(* Logix 5000 project; controller reports 1756-L63 rev 20.11; software revision 20.04; part 31 of 52 *)

        [2319].log_data[10].valid := 1, [2319].log_data[11].valid := 1, [2319].log_data[12].valid := 1, [2319].log_data[13].valid := 1, [2319].log_data[14].valid := 1, [2319].log_data[15].valid := 1, [2319].log_data[16].valid := 1, [2319].log_data[17].valid := 1, [2319].log_data[18].valid := 1, [2319].log_data[19].valid := 1, [2319].time.Year := 2023, [2319].time.Month := 1, [2319].time.Day := 17, [2319].time.Hour := 17, [2319].time.Minute := 39, [2319].time.Second := 59, [2320].log_data[0].min := 1.0, [2320].log_data[0].max := 1.0, [2320].log_data[0].total := 300.0, [2320].log_data[0].time := 300.0, [2320].log_data[0].minminute := 40, [2320].log_data[0].maxminute := 40, [2320].log_data[0].valid := 1, [2320].log_data[1].valid := 1, [2320].log_data[2].valid := 1, [2320].log_data[3].valid := 1, [2320].log_data[4].valid := 1, [2320].log_data[5].valid := 1, [2320].log_data[6].valid := 1, [2320].log_data[7].valid := 1, [2320].log_data[8].valid := 1, [2320].log_data[9].valid := 1, [2320].log_data[10].valid := 1, [2320].log_data[11].valid := 1, [2320].log_data[12].valid := 1, [2320].log_data[13].valid := 1, [2320].log_data[14].valid := 1, [2320].log_data[15].valid := 1, [2320].log_data[16].valid := 1, [2320].log_data[17].valid := 1, [2320].log_data[18].valid := 1, [2320].log_data[19].valid := 1, [2320].time.Year := 2023, [2320].time.Month := 1, [2320].time.Day := 17, [2320].time.Hour := 17, [2320].time.Minute := 44, [2320].time.Second := 59, [2321].log_data[0].min := 1.0, [2321].log_data[0].max := 1.0, [2321].log_data[0].total := 300.0, [2321].log_data[0].time := 300.0, [2321].log_data[0].minminute := 45, [2321].log_data[0].maxminute := 45, [2321].log_data[0].valid := 1, [2321].log_data[1].valid := 1, [2321].log_data[2].valid := 1, [2321].log_data[3].valid := 1, [2321].log_data[4].valid := 1, [2321].log_data[5].valid := 1,
        [2321].log_data[6].valid := 1, [2321].log_data[7].valid := 1, [2321].log_data[8].valid := 1, [2321].log_data[9].valid := 1, [2321].log_data[10].valid := 1, [2321].log_data[11].valid := 1, [2321].log_data[12].valid := 1, [2321].log_data[13].valid := 1, [2321].log_data[14].valid := 1, [2321].log_data[15].valid := 1, [2321].log_data[16].valid := 1, [2321].log_data[17].valid := 1, [2321].log_data[18].valid := 1, [2321].log_data[19].valid := 1, [2321].time.Year := 2023, [2321].time.Month := 1, [2321].time.Day := 17, [2321].time.Hour := 17, [2321].time.Minute := 49, [2321].time.Second := 59, [2322].log_data[0].min := 1.0, [2322].log_data[0].max := 1.0, [2322].log_data[0].total := 300.0, [2322].log_data[0].time := 300.0, [2322].log_data[0].minminute := 50, [2322].log_data[0].maxminute := 50, [2322].log_data[0].valid := 1, [2322].log_data[1].valid := 1, [2322].log_data[2].valid := 1, [2322].log_data[3].valid := 1, [2322].log_data[4].valid := 1, [2322].log_data[5].valid := 1, [2322].log_data[6].valid := 1, [2322].log_data[7].valid := 1, [2322].log_data[8].valid := 1, [2322].log_data[9].valid := 1, [2322].log_data[10].valid := 1, [2322].log_data[11].valid := 1, [2322].log_data[12].valid := 1, [2322].log_data[13].valid := 1, [2322].log_data[14].valid := 1, [2322].log_data[15].valid := 1, [2322].log_data[16].valid := 1, [2322].log_data[17].valid := 1, [2322].log_data[18].valid := 1, [2322].log_data[19].valid := 1, [2322].time.Year := 2023, [2322].time.Month := 1, [2322].time.Day := 17, [2322].time.Hour := 17, [2322].time.Minute := 54, [2322].time.Second := 59, [2323].log_data[0].min := 1.0, [2323].log_data[0].max := 1.0, [2323].log_data[0].total := 300.0, [2323].log_data[0].time := 300.0, [2323].log_data[0].minminute := 55, [2323].log_data[0].maxminute := 55, [2323].log_data[0].valid := 1, [2323].log_data[1].valid := 1,
        [2323].log_data[2].valid := 1, [2323].log_data[3].valid := 1, [2323].log_data[4].valid := 1, [2323].log_data[5].valid := 1, [2323].log_data[6].valid := 1, [2323].log_data[7].valid := 1, [2323].log_data[8].valid := 1, [2323].log_data[9].valid := 1, [2323].log_data[10].valid := 1, [2323].log_data[11].valid := 1, [2323].log_data[12].valid := 1, [2323].log_data[13].valid := 1, [2323].log_data[14].valid := 1, [2323].log_data[15].valid := 1, [2323].log_data[16].valid := 1, [2323].log_data[17].valid := 1, [2323].log_data[18].valid := 1, [2323].log_data[19].valid := 1, [2323].time.Year := 2023, [2323].time.Month := 1, [2323].time.Day := 17, [2323].time.Hour := 17, [2323].time.Minute := 59, [2323].time.Second := 59, [2324].log_data[0].min := 1.0, [2324].log_data[0].max := 1.0, [2324].log_data[0].total := 300.0, [2324].log_data[0].time := 300.0, [2324].log_data[0].valid := 1, [2324].log_data[1].valid := 1, [2324].log_data[2].valid := 1, [2324].log_data[3].valid := 1, [2324].log_data[4].valid := 1, [2324].log_data[5].valid := 1, [2324].log_data[6].valid := 1, [2324].log_data[7].valid := 1, [2324].log_data[8].valid := 1, [2324].log_data[9].valid := 1, [2324].log_data[10].valid := 1, [2324].log_data[11].valid := 1, [2324].log_data[12].valid := 1, [2324].log_data[13].valid := 1, [2324].log_data[14].valid := 1, [2324].log_data[15].valid := 1, [2324].log_data[16].valid := 1, [2324].log_data[17].valid := 1, [2324].log_data[18].valid := 1, [2324].log_data[19].valid := 1, [2324].time.Year := 2023, [2324].time.Month := 1, [2324].time.Day := 17, [2324].time.Hour := 18, [2324].time.Minute := 4, [2324].time.Second := 59, [2325].log_data[0].min := 1.0, [2325].log_data[0].max := 1.0, [2325].log_data[0].total := 300.0, [2325].log_data[0].time := 300.0, [2325].log_data[0].minminute := 5, [2325].log_data[0].maxminute := 5,
        [2325].log_data[0].valid := 1, [2325].log_data[1].valid := 1, [2325].log_data[2].valid := 1, [2325].log_data[3].valid := 1, [2325].log_data[4].valid := 1, [2325].log_data[5].valid := 1, [2325].log_data[6].valid := 1, [2325].log_data[7].valid := 1, [2325].log_data[8].valid := 1, [2325].log_data[9].valid := 1, [2325].log_data[10].valid := 1, [2325].log_data[11].valid := 1, [2325].log_data[12].valid := 1, [2325].log_data[13].valid := 1, [2325].log_data[14].valid := 1, [2325].log_data[15].valid := 1, [2325].log_data[16].valid := 1, [2325].log_data[17].valid := 1, [2325].log_data[18].valid := 1, [2325].log_data[19].valid := 1, [2325].time.Year := 2023, [2325].time.Month := 1, [2325].time.Day := 17, [2325].time.Hour := 18, [2325].time.Minute := 9, [2325].time.Second := 59, [2326].log_data[0].min := 1.0, [2326].log_data[0].max := 1.0, [2326].log_data[0].total := 300.0, [2326].log_data[0].time := 300.0, [2326].log_data[0].minminute := 10, [2326].log_data[0].maxminute := 10, [2326].log_data[0].valid := 1, [2326].log_data[1].valid := 1, [2326].log_data[2].valid := 1, [2326].log_data[3].valid := 1, [2326].log_data[4].valid := 1, [2326].log_data[5].valid := 1, [2326].log_data[6].valid := 1, [2326].log_data[7].valid := 1, [2326].log_data[8].valid := 1, [2326].log_data[9].valid := 1, [2326].log_data[10].valid := 1, [2326].log_data[11].valid := 1, [2326].log_data[12].valid := 1, [2326].log_data[13].valid := 1, [2326].log_data[14].valid := 1, [2326].log_data[15].valid := 1, [2326].log_data[16].valid := 1, [2326].log_data[17].valid := 1, [2326].log_data[18].valid := 1, [2326].log_data[19].valid := 1, [2326].time.Year := 2023, [2326].time.Month := 1, [2326].time.Day := 17, [2326].time.Hour := 18, [2326].time.Minute := 14, [2326].time.Second := 59, [2327].log_data[0].min := 1.0, [2327].log_data[0].max := 1.0,
        [2327].log_data[0].total := 300.0, [2327].log_data[0].time := 300.0, [2327].log_data[0].minminute := 15, [2327].log_data[0].maxminute := 15, [2327].log_data[0].valid := 1, [2327].log_data[1].valid := 1, [2327].log_data[2].valid := 1, [2327].log_data[3].valid := 1, [2327].log_data[4].valid := 1, [2327].log_data[5].valid := 1, [2327].log_data[6].valid := 1, [2327].log_data[7].valid := 1, [2327].log_data[8].valid := 1, [2327].log_data[9].valid := 1, [2327].log_data[10].valid := 1, [2327].log_data[11].valid := 1, [2327].log_data[12].valid := 1, [2327].log_data[13].valid := 1, [2327].log_data[14].valid := 1, [2327].log_data[15].valid := 1, [2327].log_data[16].valid := 1, [2327].log_data[17].valid := 1, [2327].log_data[18].valid := 1, [2327].log_data[19].valid := 1, [2327].time.Year := 2023, [2327].time.Month := 1, [2327].time.Day := 17, [2327].time.Hour := 18, [2327].time.Minute := 19, [2327].time.Second := 59, [2328].log_data[0].min := 1.0, [2328].log_data[0].max := 1.0, [2328].log_data[0].total := 300.0, [2328].log_data[0].time := 300.0, [2328].log_data[0].minminute := 20, [2328].log_data[0].maxminute := 20, [2328].log_data[0].valid := 1, [2328].log_data[1].valid := 1, [2328].log_data[2].valid := 1, [2328].log_data[3].valid := 1, [2328].log_data[4].valid := 1, [2328].log_data[5].valid := 1, [2328].log_data[6].valid := 1, [2328].log_data[7].valid := 1, [2328].log_data[8].valid := 1, [2328].log_data[9].valid := 1, [2328].log_data[10].valid := 1, [2328].log_data[11].valid := 1, [2328].log_data[12].valid := 1, [2328].log_data[13].valid := 1, [2328].log_data[14].valid := 1, [2328].log_data[15].valid := 1, [2328].log_data[16].valid := 1, [2328].log_data[17].valid := 1, [2328].log_data[18].valid := 1, [2328].log_data[19].valid := 1, [2328].time.Year := 2023, [2328].time.Month := 1, [2328].time.Day := 17, [2328].time.Hour := 18,
        [2328].time.Minute := 24, [2328].time.Second := 59, [2329].log_data[0].min := 1.0, [2329].log_data[0].max := 1.0, [2329].log_data[0].total := 300.0, [2329].log_data[0].time := 300.0, [2329].log_data[0].minminute := 25, [2329].log_data[0].maxminute := 25, [2329].log_data[0].valid := 1, [2329].log_data[1].valid := 1, [2329].log_data[2].valid := 1, [2329].log_data[3].valid := 1, [2329].log_data[4].valid := 1, [2329].log_data[5].valid := 1, [2329].log_data[6].valid := 1, [2329].log_data[7].valid := 1, [2329].log_data[8].valid := 1, [2329].log_data[9].valid := 1, [2329].log_data[10].valid := 1, [2329].log_data[11].valid := 1, [2329].log_data[12].valid := 1, [2329].log_data[13].valid := 1, [2329].log_data[14].valid := 1, [2329].log_data[15].valid := 1, [2329].log_data[16].valid := 1, [2329].log_data[17].valid := 1, [2329].log_data[18].valid := 1, [2329].log_data[19].valid := 1, [2329].time.Year := 2023, [2329].time.Month := 1, [2329].time.Day := 17, [2329].time.Hour := 18, [2329].time.Minute := 29, [2329].time.Second := 59, [2330].log_data[0].min := 1.0, [2330].log_data[0].max := 1.0, [2330].log_data[0].total := 300.0, [2330].log_data[0].time := 300.0, [2330].log_data[0].minminute := 30, [2330].log_data[0].maxminute := 30, [2330].log_data[0].valid := 1, [2330].log_data[1].valid := 1, [2330].log_data[2].valid := 1, [2330].log_data[3].valid := 1, [2330].log_data[4].valid := 1, [2330].log_data[5].valid := 1, [2330].log_data[6].valid := 1, [2330].log_data[7].valid := 1, [2330].log_data[8].valid := 1, [2330].log_data[9].valid := 1, [2330].log_data[10].valid := 1, [2330].log_data[11].valid := 1, [2330].log_data[12].valid := 1, [2330].log_data[13].valid := 1, [2330].log_data[14].valid := 1, [2330].log_data[15].valid := 1, [2330].log_data[16].valid := 1, [2330].log_data[17].valid := 1, [2330].log_data[18].valid := 1, [2330].log_data[19].valid := 1,
        [2330].time.Year := 2023, [2330].time.Month := 1, [2330].time.Day := 17, [2330].time.Hour := 18, [2330].time.Minute := 34, [2330].time.Second := 59, [2331].log_data[0].min := 1.0, [2331].log_data[0].max := 1.0, [2331].log_data[0].total := 300.0, [2331].log_data[0].time := 300.0, [2331].log_data[0].minminute := 35, [2331].log_data[0].maxminute := 35, [2331].log_data[0].valid := 1, [2331].log_data[1].valid := 1, [2331].log_data[2].valid := 1, [2331].log_data[3].valid := 1, [2331].log_data[4].valid := 1, [2331].log_data[5].valid := 1, [2331].log_data[6].valid := 1, [2331].log_data[7].valid := 1, [2331].log_data[8].valid := 1, [2331].log_data[9].valid := 1, [2331].log_data[10].valid := 1, [2331].log_data[11].valid := 1, [2331].log_data[12].valid := 1, [2331].log_data[13].valid := 1, [2331].log_data[14].valid := 1, [2331].log_data[15].valid := 1, [2331].log_data[16].valid := 1, [2331].log_data[17].valid := 1, [2331].log_data[18].valid := 1, [2331].log_data[19].valid := 1, [2331].time.Year := 2023, [2331].time.Month := 1, [2331].time.Day := 17, [2331].time.Hour := 18, [2331].time.Minute := 39, [2331].time.Second := 59, [2332].log_data[0].min := 1.0, [2332].log_data[0].max := 1.0, [2332].log_data[0].total := 300.0, [2332].log_data[0].time := 300.0, [2332].log_data[0].minminute := 40, [2332].log_data[0].maxminute := 40, [2332].log_data[0].valid := 1, [2332].log_data[1].valid := 1, [2332].log_data[2].valid := 1, [2332].log_data[3].valid := 1, [2332].log_data[4].valid := 1, [2332].log_data[5].valid := 1, [2332].log_data[6].valid := 1, [2332].log_data[7].valid := 1, [2332].log_data[8].valid := 1, [2332].log_data[9].valid := 1, [2332].log_data[10].valid := 1, [2332].log_data[11].valid := 1, [2332].log_data[12].valid := 1, [2332].log_data[13].valid := 1, [2332].log_data[14].valid := 1, [2332].log_data[15].valid := 1,
        [2332].log_data[16].valid := 1, [2332].log_data[17].valid := 1, [2332].log_data[18].valid := 1, [2332].log_data[19].valid := 1, [2332].time.Year := 2023, [2332].time.Month := 1, [2332].time.Day := 17, [2332].time.Hour := 18, [2332].time.Minute := 44, [2332].time.Second := 59, [2333].log_data[0].min := 1.0, [2333].log_data[0].max := 1.0, [2333].log_data[0].total := 300.0, [2333].log_data[0].time := 300.0, [2333].log_data[0].minminute := 45, [2333].log_data[0].maxminute := 45, [2333].log_data[0].valid := 1, [2333].log_data[1].valid := 1, [2333].log_data[2].valid := 1, [2333].log_data[3].valid := 1, [2333].log_data[4].valid := 1, [2333].log_data[5].valid := 1, [2333].log_data[6].valid := 1, [2333].log_data[7].valid := 1, [2333].log_data[8].valid := 1, [2333].log_data[9].valid := 1, [2333].log_data[10].valid := 1, [2333].log_data[11].valid := 1, [2333].log_data[12].valid := 1, [2333].log_data[13].valid := 1, [2333].log_data[14].valid := 1, [2333].log_data[15].valid := 1, [2333].log_data[16].valid := 1, [2333].log_data[17].valid := 1, [2333].log_data[18].valid := 1, [2333].log_data[19].valid := 1, [2333].time.Year := 2023, [2333].time.Month := 1, [2333].time.Day := 17, [2333].time.Hour := 18, [2333].time.Minute := 49, [2333].time.Second := 59, [2334].log_data[0].min := 1.0, [2334].log_data[0].max := 1.0, [2334].log_data[0].total := 300.0, [2334].log_data[0].time := 300.0, [2334].log_data[0].minminute := 50, [2334].log_data[0].maxminute := 50, [2334].log_data[0].valid := 1, [2334].log_data[1].valid := 1, [2334].log_data[2].valid := 1, [2334].log_data[3].valid := 1, [2334].log_data[4].valid := 1, [2334].log_data[5].valid := 1, [2334].log_data[6].valid := 1, [2334].log_data[7].valid := 1, [2334].log_data[8].valid := 1, [2334].log_data[9].valid := 1, [2334].log_data[10].valid := 1, [2334].log_data[11].valid := 1,
        [2334].log_data[12].valid := 1, [2334].log_data[13].valid := 1, [2334].log_data[14].valid := 1, [2334].log_data[15].valid := 1, [2334].log_data[16].valid := 1, [2334].log_data[17].valid := 1, [2334].log_data[18].valid := 1, [2334].log_data[19].valid := 1, [2334].time.Year := 2023, [2334].time.Month := 1, [2334].time.Day := 17, [2334].time.Hour := 18, [2334].time.Minute := 54, [2334].time.Second := 59, [2335].log_data[0].min := 1.0, [2335].log_data[0].max := 1.0, [2335].log_data[0].total := 300.0, [2335].log_data[0].time := 300.0, [2335].log_data[0].minminute := 55, [2335].log_data[0].maxminute := 55, [2335].log_data[0].valid := 1, [2335].log_data[1].valid := 1, [2335].log_data[2].valid := 1, [2335].log_data[3].valid := 1, [2335].log_data[4].valid := 1, [2335].log_data[5].valid := 1, [2335].log_data[6].valid := 1, [2335].log_data[7].valid := 1, [2335].log_data[8].valid := 1, [2335].log_data[9].valid := 1, [2335].log_data[10].valid := 1, [2335].log_data[11].valid := 1, [2335].log_data[12].valid := 1, [2335].log_data[13].valid := 1, [2335].log_data[14].valid := 1, [2335].log_data[15].valid := 1, [2335].log_data[16].valid := 1, [2335].log_data[17].valid := 1, [2335].log_data[18].valid := 1, [2335].log_data[19].valid := 1, [2335].time.Year := 2023, [2335].time.Month := 1, [2335].time.Day := 17, [2335].time.Hour := 18, [2335].time.Minute := 59, [2335].time.Second := 59, [2336].log_data[0].min := 1.0, [2336].log_data[0].max := 1.0, [2336].log_data[0].total := 300.0, [2336].log_data[0].time := 300.0, [2336].log_data[0].valid := 1, [2336].log_data[1].valid := 1, [2336].log_data[2].valid := 1, [2336].log_data[3].valid := 1, [2336].log_data[4].valid := 1, [2336].log_data[5].valid := 1, [2336].log_data[6].valid := 1, [2336].log_data[7].valid := 1, [2336].log_data[8].valid := 1, [2336].log_data[9].valid := 1,
        [2336].log_data[10].valid := 1, [2336].log_data[11].valid := 1, [2336].log_data[12].valid := 1, [2336].log_data[13].valid := 1, [2336].log_data[14].valid := 1, [2336].log_data[15].valid := 1, [2336].log_data[16].valid := 1, [2336].log_data[17].valid := 1, [2336].log_data[18].valid := 1, [2336].log_data[19].valid := 1, [2336].time.Year := 2023, [2336].time.Month := 1, [2336].time.Day := 17, [2336].time.Hour := 19, [2336].time.Minute := 4, [2336].time.Second := 59, [2337].log_data[0].min := 1.0, [2337].log_data[0].max := 1.0, [2337].log_data[0].total := 300.0, [2337].log_data[0].time := 300.0, [2337].log_data[0].minminute := 5, [2337].log_data[0].maxminute := 5, [2337].log_data[0].valid := 1, [2337].log_data[1].valid := 1, [2337].log_data[2].valid := 1, [2337].log_data[3].valid := 1, [2337].log_data[4].valid := 1, [2337].log_data[5].valid := 1, [2337].log_data[6].valid := 1, [2337].log_data[7].valid := 1, [2337].log_data[8].valid := 1, [2337].log_data[9].valid := 1, [2337].log_data[10].valid := 1, [2337].log_data[11].valid := 1, [2337].log_data[12].valid := 1, [2337].log_data[13].valid := 1, [2337].log_data[14].valid := 1, [2337].log_data[15].valid := 1, [2337].log_data[16].valid := 1, [2337].log_data[17].valid := 1, [2337].log_data[18].valid := 1, [2337].log_data[19].valid := 1, [2337].time.Year := 2023, [2337].time.Month := 1, [2337].time.Day := 17, [2337].time.Hour := 19, [2337].time.Minute := 9, [2337].time.Second := 59, [2338].log_data[0].min := 1.0, [2338].log_data[0].max := 1.0, [2338].log_data[0].total := 300.0, [2338].log_data[0].time := 300.0, [2338].log_data[0].minminute := 10, [2338].log_data[0].maxminute := 10, [2338].log_data[0].valid := 1, [2338].log_data[1].valid := 1, [2338].log_data[2].valid := 1, [2338].log_data[3].valid := 1, [2338].log_data[4].valid := 1, [2338].log_data[5].valid := 1,
        [2338].log_data[6].valid := 1, [2338].log_data[7].valid := 1, [2338].log_data[8].valid := 1, [2338].log_data[9].valid := 1, [2338].log_data[10].valid := 1, [2338].log_data[11].valid := 1, [2338].log_data[12].valid := 1, [2338].log_data[13].valid := 1, [2338].log_data[14].valid := 1, [2338].log_data[15].valid := 1, [2338].log_data[16].valid := 1, [2338].log_data[17].valid := 1, [2338].log_data[18].valid := 1, [2338].log_data[19].valid := 1, [2338].time.Year := 2023, [2338].time.Month := 1, [2338].time.Day := 17, [2338].time.Hour := 19, [2338].time.Minute := 14, [2338].time.Second := 59, [2339].log_data[0].min := 1.0, [2339].log_data[0].max := 1.0, [2339].log_data[0].total := 300.0, [2339].log_data[0].time := 300.0, [2339].log_data[0].minminute := 15, [2339].log_data[0].maxminute := 15, [2339].log_data[0].valid := 1, [2339].log_data[1].valid := 1, [2339].log_data[2].valid := 1, [2339].log_data[3].valid := 1, [2339].log_data[4].valid := 1, [2339].log_data[5].valid := 1, [2339].log_data[6].valid := 1, [2339].log_data[7].valid := 1, [2339].log_data[8].valid := 1, [2339].log_data[9].valid := 1, [2339].log_data[10].valid := 1, [2339].log_data[11].valid := 1, [2339].log_data[12].valid := 1, [2339].log_data[13].valid := 1, [2339].log_data[14].valid := 1, [2339].log_data[15].valid := 1, [2339].log_data[16].valid := 1, [2339].log_data[17].valid := 1, [2339].log_data[18].valid := 1, [2339].log_data[19].valid := 1, [2339].time.Year := 2023, [2339].time.Month := 1, [2339].time.Day := 17, [2339].time.Hour := 19, [2339].time.Minute := 19, [2339].time.Second := 59, [2340].log_data[0].min := 1.0, [2340].log_data[0].max := 1.0, [2340].log_data[0].total := 300.0, [2340].log_data[0].time := 300.0, [2340].log_data[0].minminute := 20, [2340].log_data[0].maxminute := 20, [2340].log_data[0].valid := 1, [2340].log_data[1].valid := 1,
        [2340].log_data[2].valid := 1, [2340].log_data[3].valid := 1, [2340].log_data[4].valid := 1, [2340].log_data[5].valid := 1, [2340].log_data[6].valid := 1, [2340].log_data[7].valid := 1, [2340].log_data[8].valid := 1, [2340].log_data[9].valid := 1, [2340].log_data[10].valid := 1, [2340].log_data[11].valid := 1, [2340].log_data[12].valid := 1, [2340].log_data[13].valid := 1, [2340].log_data[14].valid := 1, [2340].log_data[15].valid := 1, [2340].log_data[16].valid := 1, [2340].log_data[17].valid := 1, [2340].log_data[18].valid := 1, [2340].log_data[19].valid := 1, [2340].time.Year := 2023, [2340].time.Month := 1, [2340].time.Day := 17, [2340].time.Hour := 19, [2340].time.Minute := 24, [2340].time.Second := 59, [2341].log_data[0].min := 1.0, [2341].log_data[0].max := 1.0, [2341].log_data[0].total := 300.0, [2341].log_data[0].time := 300.0, [2341].log_data[0].minminute := 25, [2341].log_data[0].maxminute := 25, [2341].log_data[0].valid := 1, [2341].log_data[1].valid := 1, [2341].log_data[2].valid := 1, [2341].log_data[3].valid := 1, [2341].log_data[4].valid := 1, [2341].log_data[5].valid := 1, [2341].log_data[6].valid := 1, [2341].log_data[7].valid := 1, [2341].log_data[8].valid := 1, [2341].log_data[9].valid := 1, [2341].log_data[10].valid := 1, [2341].log_data[11].valid := 1, [2341].log_data[12].valid := 1, [2341].log_data[13].valid := 1, [2341].log_data[14].valid := 1, [2341].log_data[15].valid := 1, [2341].log_data[16].valid := 1, [2341].log_data[17].valid := 1, [2341].log_data[18].valid := 1, [2341].log_data[19].valid := 1, [2341].time.Year := 2023, [2341].time.Month := 1, [2341].time.Day := 17, [2341].time.Hour := 19, [2341].time.Minute := 29, [2341].time.Second := 59, [2342].log_data[0].min := 1.0, [2342].log_data[0].max := 1.0, [2342].log_data[0].total := 300.0, [2342].log_data[0].time := 300.0,
        [2342].log_data[0].minminute := 30, [2342].log_data[0].maxminute := 30, [2342].log_data[0].valid := 1, [2342].log_data[1].valid := 1, [2342].log_data[2].valid := 1, [2342].log_data[3].valid := 1, [2342].log_data[4].valid := 1, [2342].log_data[5].valid := 1, [2342].log_data[6].valid := 1, [2342].log_data[7].valid := 1, [2342].log_data[8].valid := 1, [2342].log_data[9].valid := 1, [2342].log_data[10].valid := 1, [2342].log_data[11].valid := 1, [2342].log_data[12].valid := 1, [2342].log_data[13].valid := 1, [2342].log_data[14].valid := 1, [2342].log_data[15].valid := 1, [2342].log_data[16].valid := 1, [2342].log_data[17].valid := 1, [2342].log_data[18].valid := 1, [2342].log_data[19].valid := 1, [2342].time.Year := 2023, [2342].time.Month := 1, [2342].time.Day := 17, [2342].time.Hour := 19, [2342].time.Minute := 34, [2342].time.Second := 59, [2343].log_data[0].min := 1.0, [2343].log_data[0].max := 1.0, [2343].log_data[0].total := 300.0, [2343].log_data[0].time := 300.0, [2343].log_data[0].minminute := 35, [2343].log_data[0].maxminute := 35, [2343].log_data[0].valid := 1, [2343].log_data[1].valid := 1, [2343].log_data[2].valid := 1, [2343].log_data[3].valid := 1, [2343].log_data[4].valid := 1, [2343].log_data[5].valid := 1, [2343].log_data[6].valid := 1, [2343].log_data[7].valid := 1, [2343].log_data[8].valid := 1, [2343].log_data[9].valid := 1, [2343].log_data[10].valid := 1, [2343].log_data[11].valid := 1, [2343].log_data[12].valid := 1, [2343].log_data[13].valid := 1, [2343].log_data[14].valid := 1, [2343].log_data[15].valid := 1, [2343].log_data[16].valid := 1, [2343].log_data[17].valid := 1, [2343].log_data[18].valid := 1, [2343].log_data[19].valid := 1, [2343].time.Year := 2023, [2343].time.Month := 1, [2343].time.Day := 17, [2343].time.Hour := 19, [2343].time.Minute := 39, [2343].time.Second := 59,
        [2344].log_data[0].min := 1.0, [2344].log_data[0].max := 1.0, [2344].log_data[0].total := 300.0, [2344].log_data[0].time := 300.0, [2344].log_data[0].minminute := 40, [2344].log_data[0].maxminute := 40, [2344].log_data[0].valid := 1, [2344].log_data[1].valid := 1, [2344].log_data[2].valid := 1, [2344].log_data[3].valid := 1, [2344].log_data[4].valid := 1, [2344].log_data[5].valid := 1, [2344].log_data[6].valid := 1, [2344].log_data[7].valid := 1, [2344].log_data[8].valid := 1, [2344].log_data[9].valid := 1, [2344].log_data[10].valid := 1, [2344].log_data[11].valid := 1, [2344].log_data[12].valid := 1, [2344].log_data[13].valid := 1, [2344].log_data[14].valid := 1, [2344].log_data[15].valid := 1, [2344].log_data[16].valid := 1, [2344].log_data[17].valid := 1, [2344].log_data[18].valid := 1, [2344].log_data[19].valid := 1, [2344].time.Year := 2023, [2344].time.Month := 1, [2344].time.Day := 17, [2344].time.Hour := 19, [2344].time.Minute := 44, [2344].time.Second := 59, [2345].log_data[0].min := 1.0, [2345].log_data[0].max := 1.0, [2345].log_data[0].total := 300.0, [2345].log_data[0].time := 300.0, [2345].log_data[0].minminute := 45, [2345].log_data[0].maxminute := 45, [2345].log_data[0].valid := 1, [2345].log_data[1].valid := 1, [2345].log_data[2].valid := 1, [2345].log_data[3].valid := 1, [2345].log_data[4].valid := 1, [2345].log_data[5].valid := 1, [2345].log_data[6].valid := 1, [2345].log_data[7].valid := 1, [2345].log_data[8].valid := 1, [2345].log_data[9].valid := 1, [2345].log_data[10].valid := 1, [2345].log_data[11].valid := 1, [2345].log_data[12].valid := 1, [2345].log_data[13].valid := 1, [2345].log_data[14].valid := 1, [2345].log_data[15].valid := 1, [2345].log_data[16].valid := 1, [2345].log_data[17].valid := 1, [2345].log_data[18].valid := 1, [2345].log_data[19].valid := 1, [2345].time.Year := 2023, [2345].time.Month := 1,
        [2345].time.Day := 17, [2345].time.Hour := 19, [2345].time.Minute := 49, [2345].time.Second := 59, [2346].log_data[0].min := 1.0, [2346].log_data[0].max := 1.0, [2346].log_data[0].total := 300.0, [2346].log_data[0].time := 300.0, [2346].log_data[0].minminute := 50, [2346].log_data[0].maxminute := 50, [2346].log_data[0].valid := 1, [2346].log_data[1].valid := 1, [2346].log_data[2].valid := 1, [2346].log_data[3].valid := 1, [2346].log_data[4].valid := 1, [2346].log_data[5].valid := 1, [2346].log_data[6].valid := 1, [2346].log_data[7].valid := 1, [2346].log_data[8].valid := 1, [2346].log_data[9].valid := 1, [2346].log_data[10].valid := 1, [2346].log_data[11].valid := 1, [2346].log_data[12].valid := 1, [2346].log_data[13].valid := 1, [2346].log_data[14].valid := 1, [2346].log_data[15].valid := 1, [2346].log_data[16].valid := 1, [2346].log_data[17].valid := 1, [2346].log_data[18].valid := 1, [2346].log_data[19].valid := 1, [2346].time.Year := 2023, [2346].time.Month := 1, [2346].time.Day := 17, [2346].time.Hour := 19, [2346].time.Minute := 54, [2346].time.Second := 59, [2347].log_data[0].min := 1.0, [2347].log_data[0].max := 1.0, [2347].log_data[0].total := 300.0, [2347].log_data[0].time := 300.0, [2347].log_data[0].minminute := 55, [2347].log_data[0].maxminute := 55, [2347].log_data[0].valid := 1, [2347].log_data[1].valid := 1, [2347].log_data[2].valid := 1, [2347].log_data[3].valid := 1, [2347].log_data[4].valid := 1, [2347].log_data[5].valid := 1, [2347].log_data[6].valid := 1, [2347].log_data[7].valid := 1, [2347].log_data[8].valid := 1, [2347].log_data[9].valid := 1, [2347].log_data[10].valid := 1, [2347].log_data[11].valid := 1, [2347].log_data[12].valid := 1, [2347].log_data[13].valid := 1, [2347].log_data[14].valid := 1, [2347].log_data[15].valid := 1, [2347].log_data[16].valid := 1, [2347].log_data[17].valid := 1,
        [2347].log_data[18].valid := 1, [2347].log_data[19].valid := 1, [2347].time.Year := 2023, [2347].time.Month := 1, [2347].time.Day := 17, [2347].time.Hour := 19, [2347].time.Minute := 59, [2347].time.Second := 59, [2348].log_data[0].min := 1.0, [2348].log_data[0].max := 1.0, [2348].log_data[0].total := 299.5, [2348].log_data[0].time := 299.5, [2348].log_data[0].valid := 1, [2348].log_data[1].valid := 1, [2348].log_data[2].valid := 1, [2348].log_data[3].valid := 1, [2348].log_data[4].valid := 1, [2348].log_data[5].valid := 1, [2348].log_data[6].valid := 1, [2348].log_data[7].valid := 1, [2348].log_data[8].valid := 1, [2348].log_data[9].valid := 1, [2348].log_data[10].valid := 1, [2348].log_data[11].valid := 1, [2348].log_data[12].valid := 1, [2348].log_data[13].valid := 1, [2348].log_data[14].valid := 1, [2348].log_data[15].valid := 1, [2348].log_data[16].valid := 1, [2348].log_data[17].valid := 1, [2348].log_data[18].valid := 1, [2348].log_data[19].valid := 1, [2348].time.Year := 2023, [2348].time.Month := 1, [2348].time.Day := 17, [2348].time.Hour := 20, [2348].time.Minute := 4, [2348].time.Second := 59, [2349].log_data[0].min := 1.0, [2349].log_data[0].max := 1.0, [2349].log_data[0].total := 300.0, [2349].log_data[0].time := 300.0, [2349].log_data[0].minminute := 5, [2349].log_data[0].maxminute := 5, [2349].log_data[0].valid := 1, [2349].log_data[1].valid := 1, [2349].log_data[2].valid := 1, [2349].log_data[3].valid := 1, [2349].log_data[4].valid := 1, [2349].log_data[5].valid := 1, [2349].log_data[6].valid := 1, [2349].log_data[7].valid := 1, [2349].log_data[8].valid := 1, [2349].log_data[9].valid := 1, [2349].log_data[10].valid := 1, [2349].log_data[11].valid := 1, [2349].log_data[12].valid := 1, [2349].log_data[13].valid := 1, [2349].log_data[14].valid := 1, [2349].log_data[15].valid := 1,
        [2349].log_data[16].valid := 1, [2349].log_data[17].valid := 1, [2349].log_data[18].valid := 1, [2349].log_data[19].valid := 1, [2349].time.Year := 2023, [2349].time.Month := 1, [2349].time.Day := 17, [2349].time.Hour := 20, [2349].time.Minute := 9, [2349].time.Second := 59, [2350].log_data[0].min := 1.0, [2350].log_data[0].max := 1.0, [2350].log_data[0].total := 300.0, [2350].log_data[0].time := 300.0, [2350].log_data[0].minminute := 10, [2350].log_data[0].maxminute := 10, [2350].log_data[0].valid := 1, [2350].log_data[1].valid := 1, [2350].log_data[2].valid := 1, [2350].log_data[3].valid := 1, [2350].log_data[4].valid := 1, [2350].log_data[5].valid := 1, [2350].log_data[6].valid := 1, [2350].log_data[7].valid := 1, [2350].log_data[8].valid := 1, [2350].log_data[9].valid := 1, [2350].log_data[10].valid := 1, [2350].log_data[11].valid := 1, [2350].log_data[12].valid := 1, [2350].log_data[13].valid := 1, [2350].log_data[14].valid := 1, [2350].log_data[15].valid := 1, [2350].log_data[16].valid := 1, [2350].log_data[17].valid := 1, [2350].log_data[18].valid := 1, [2350].log_data[19].valid := 1, [2350].time.Year := 2023, [2350].time.Month := 1, [2350].time.Day := 17, [2350].time.Hour := 20, [2350].time.Minute := 14, [2350].time.Second := 59, [2351].log_data[0].min := 1.0, [2351].log_data[0].max := 1.0, [2351].log_data[0].total := 300.0, [2351].log_data[0].time := 300.0, [2351].log_data[0].minminute := 15, [2351].log_data[0].maxminute := 15, [2351].log_data[0].valid := 1, [2351].log_data[1].valid := 1, [2351].log_data[2].valid := 1, [2351].log_data[3].valid := 1, [2351].log_data[4].valid := 1, [2351].log_data[5].valid := 1, [2351].log_data[6].valid := 1, [2351].log_data[7].valid := 1, [2351].log_data[8].valid := 1, [2351].log_data[9].valid := 1, [2351].log_data[10].valid := 1, [2351].log_data[11].valid := 1,
        [2351].log_data[12].valid := 1, [2351].log_data[13].valid := 1, [2351].log_data[14].valid := 1, [2351].log_data[15].valid := 1, [2351].log_data[16].valid := 1, [2351].log_data[17].valid := 1, [2351].log_data[18].valid := 1, [2351].log_data[19].valid := 1, [2351].time.Year := 2023, [2351].time.Month := 1, [2351].time.Day := 17, [2351].time.Hour := 20, [2351].time.Minute := 19, [2351].time.Second := 59, [2352].log_data[0].min := 1.0, [2352].log_data[0].max := 1.0, [2352].log_data[0].total := 300.0, [2352].log_data[0].time := 300.0, [2352].log_data[0].minminute := 20, [2352].log_data[0].maxminute := 20, [2352].log_data[0].valid := 1, [2352].log_data[1].valid := 1, [2352].log_data[2].valid := 1, [2352].log_data[3].valid := 1, [2352].log_data[4].valid := 1, [2352].log_data[5].valid := 1, [2352].log_data[6].valid := 1, [2352].log_data[7].valid := 1, [2352].log_data[8].valid := 1, [2352].log_data[9].valid := 1, [2352].log_data[10].valid := 1, [2352].log_data[11].valid := 1, [2352].log_data[12].valid := 1, [2352].log_data[13].valid := 1, [2352].log_data[14].valid := 1, [2352].log_data[15].valid := 1, [2352].log_data[16].valid := 1, [2352].log_data[17].valid := 1, [2352].log_data[18].valid := 1, [2352].log_data[19].valid := 1, [2352].time.Year := 2023, [2352].time.Month := 1, [2352].time.Day := 17, [2352].time.Hour := 20, [2352].time.Minute := 24, [2352].time.Second := 59, [2353].log_data[0].min := 1.0, [2353].log_data[0].max := 1.0, [2353].log_data[0].total := 300.0, [2353].log_data[0].time := 300.0, [2353].log_data[0].minminute := 25, [2353].log_data[0].maxminute := 25, [2353].log_data[0].valid := 1, [2353].log_data[1].valid := 1, [2353].log_data[2].valid := 1, [2353].log_data[3].valid := 1, [2353].log_data[4].valid := 1, [2353].log_data[5].valid := 1, [2353].log_data[6].valid := 1, [2353].log_data[7].valid := 1,
        [2353].log_data[8].valid := 1, [2353].log_data[9].valid := 1, [2353].log_data[10].valid := 1, [2353].log_data[11].valid := 1, [2353].log_data[12].valid := 1, [2353].log_data[13].valid := 1, [2353].log_data[14].valid := 1, [2353].log_data[15].valid := 1, [2353].log_data[16].valid := 1, [2353].log_data[17].valid := 1, [2353].log_data[18].valid := 1, [2353].log_data[19].valid := 1, [2353].time.Year := 2023, [2353].time.Month := 1, [2353].time.Day := 17, [2353].time.Hour := 20, [2353].time.Minute := 29, [2353].time.Second := 59, [2354].log_data[0].min := 1.0, [2354].log_data[0].max := 1.0, [2354].log_data[0].total := 300.0, [2354].log_data[0].time := 300.0, [2354].log_data[0].minminute := 30, [2354].log_data[0].maxminute := 30, [2354].log_data[0].valid := 1, [2354].log_data[1].valid := 1, [2354].log_data[2].valid := 1, [2354].log_data[3].valid := 1, [2354].log_data[4].valid := 1, [2354].log_data[5].valid := 1, [2354].log_data[6].valid := 1, [2354].log_data[7].valid := 1, [2354].log_data[8].valid := 1, [2354].log_data[9].valid := 1, [2354].log_data[10].valid := 1, [2354].log_data[11].valid := 1, [2354].log_data[12].valid := 1, [2354].log_data[13].valid := 1, [2354].log_data[14].valid := 1, [2354].log_data[15].valid := 1, [2354].log_data[16].valid := 1, [2354].log_data[17].valid := 1, [2354].log_data[18].valid := 1, [2354].log_data[19].valid := 1, [2354].time.Year := 2023, [2354].time.Month := 1, [2354].time.Day := 17, [2354].time.Hour := 20, [2354].time.Minute := 34, [2354].time.Second := 59, [2355].log_data[0].min := 1.0, [2355].log_data[0].max := 1.0, [2355].log_data[0].total := 300.0, [2355].log_data[0].time := 300.0, [2355].log_data[0].minminute := 35, [2355].log_data[0].maxminute := 35, [2355].log_data[0].valid := 1, [2355].log_data[1].valid := 1, [2355].log_data[2].valid := 1, [2355].log_data[3].valid := 1,
        [2355].log_data[4].valid := 1, [2355].log_data[5].valid := 1, [2355].log_data[6].valid := 1, [2355].log_data[7].valid := 1, [2355].log_data[8].valid := 1, [2355].log_data[9].valid := 1, [2355].log_data[10].valid := 1, [2355].log_data[11].valid := 1, [2355].log_data[12].valid := 1, [2355].log_data[13].valid := 1, [2355].log_data[14].valid := 1, [2355].log_data[15].valid := 1, [2355].log_data[16].valid := 1, [2355].log_data[17].valid := 1, [2355].log_data[18].valid := 1, [2355].log_data[19].valid := 1, [2355].time.Year := 2023, [2355].time.Month := 1, [2355].time.Day := 17, [2355].time.Hour := 20, [2355].time.Minute := 39, [2355].time.Second := 59, [2356].log_data[0].min := 1.0, [2356].log_data[0].max := 1.0, [2356].log_data[0].total := 300.0, [2356].log_data[0].time := 300.0, [2356].log_data[0].minminute := 40, [2356].log_data[0].maxminute := 40, [2356].log_data[0].valid := 1, [2356].log_data[1].valid := 1, [2356].log_data[2].valid := 1, [2356].log_data[3].valid := 1, [2356].log_data[4].valid := 1, [2356].log_data[5].valid := 1, [2356].log_data[6].valid := 1, [2356].log_data[7].valid := 1, [2356].log_data[8].valid := 1, [2356].log_data[9].valid := 1, [2356].log_data[10].valid := 1, [2356].log_data[11].valid := 1, [2356].log_data[12].valid := 1, [2356].log_data[13].valid := 1, [2356].log_data[14].valid := 1, [2356].log_data[15].valid := 1, [2356].log_data[16].valid := 1, [2356].log_data[17].valid := 1, [2356].log_data[18].valid := 1, [2356].log_data[19].valid := 1, [2356].time.Year := 2023, [2356].time.Month := 1, [2356].time.Day := 17, [2356].time.Hour := 20, [2356].time.Minute := 44, [2356].time.Second := 59, [2357].log_data[0].min := 1.0, [2357].log_data[0].max := 1.0, [2357].log_data[0].total := 300.0, [2357].log_data[0].time := 300.0, [2357].log_data[0].minminute := 45, [2357].log_data[0].maxminute := 45,
        [2357].log_data[0].valid := 1, [2357].log_data[1].valid := 1, [2357].log_data[2].valid := 1, [2357].log_data[3].valid := 1, [2357].log_data[4].valid := 1, [2357].log_data[5].valid := 1, [2357].log_data[6].valid := 1, [2357].log_data[7].valid := 1, [2357].log_data[8].valid := 1, [2357].log_data[9].valid := 1, [2357].log_data[10].valid := 1, [2357].log_data[11].valid := 1, [2357].log_data[12].valid := 1, [2357].log_data[13].valid := 1, [2357].log_data[14].valid := 1, [2357].log_data[15].valid := 1, [2357].log_data[16].valid := 1, [2357].log_data[17].valid := 1, [2357].log_data[18].valid := 1, [2357].log_data[19].valid := 1, [2357].time.Year := 2023, [2357].time.Month := 1, [2357].time.Day := 17, [2357].time.Hour := 20, [2357].time.Minute := 49, [2357].time.Second := 59, [2358].log_data[0].min := 1.0, [2358].log_data[0].max := 1.0, [2358].log_data[0].total := 300.0, [2358].log_data[0].time := 300.0, [2358].log_data[0].minminute := 50, [2358].log_data[0].maxminute := 50, [2358].log_data[0].valid := 1, [2358].log_data[1].valid := 1, [2358].log_data[2].valid := 1, [2358].log_data[3].valid := 1, [2358].log_data[4].valid := 1, [2358].log_data[5].valid := 1, [2358].log_data[6].valid := 1, [2358].log_data[7].valid := 1, [2358].log_data[8].valid := 1, [2358].log_data[9].valid := 1, [2358].log_data[10].valid := 1, [2358].log_data[11].valid := 1, [2358].log_data[12].valid := 1, [2358].log_data[13].valid := 1, [2358].log_data[14].valid := 1, [2358].log_data[15].valid := 1, [2358].log_data[16].valid := 1, [2358].log_data[17].valid := 1, [2358].log_data[18].valid := 1, [2358].log_data[19].valid := 1, [2358].time.Year := 2023, [2358].time.Month := 1, [2358].time.Day := 17, [2358].time.Hour := 20, [2358].time.Minute := 54, [2358].time.Second := 59, [2359].log_data[0].min := 1.0, [2359].log_data[0].max := 1.0,
        [2359].log_data[0].total := 300.0, [2359].log_data[0].time := 300.0, [2359].log_data[0].minminute := 55, [2359].log_data[0].maxminute := 55, [2359].log_data[0].valid := 1, [2359].log_data[1].valid := 1, [2359].log_data[2].valid := 1, [2359].log_data[3].valid := 1, [2359].log_data[4].valid := 1, [2359].log_data[5].valid := 1, [2359].log_data[6].valid := 1, [2359].log_data[7].valid := 1, [2359].log_data[8].valid := 1, [2359].log_data[9].valid := 1, [2359].log_data[10].valid := 1, [2359].log_data[11].valid := 1, [2359].log_data[12].valid := 1, [2359].log_data[13].valid := 1, [2359].log_data[14].valid := 1, [2359].log_data[15].valid := 1, [2359].log_data[16].valid := 1, [2359].log_data[17].valid := 1, [2359].log_data[18].valid := 1, [2359].log_data[19].valid := 1, [2359].time.Year := 2023, [2359].time.Month := 1, [2359].time.Day := 17, [2359].time.Hour := 20, [2359].time.Minute := 59, [2359].time.Second := 59, [2360].log_data[0].min := 1.0, [2360].log_data[0].max := 1.0, [2360].log_data[0].total := 300.0, [2360].log_data[0].time := 300.0, [2360].log_data[0].valid := 1, [2360].log_data[1].valid := 1, [2360].log_data[2].valid := 1, [2360].log_data[3].valid := 1, [2360].log_data[4].valid := 1, [2360].log_data[5].valid := 1, [2360].log_data[6].valid := 1, [2360].log_data[7].valid := 1, [2360].log_data[8].valid := 1, [2360].log_data[9].valid := 1, [2360].log_data[10].valid := 1, [2360].log_data[11].valid := 1, [2360].log_data[12].valid := 1, [2360].log_data[13].valid := 1, [2360].log_data[14].valid := 1, [2360].log_data[15].valid := 1, [2360].log_data[16].valid := 1, [2360].log_data[17].valid := 1, [2360].log_data[18].valid := 1, [2360].log_data[19].valid := 1, [2360].time.Year := 2023, [2360].time.Month := 1, [2360].time.Day := 17, [2360].time.Hour := 21, [2360].time.Minute := 4, [2360].time.Second := 59,
        [2361].log_data[0].min := 1.0, [2361].log_data[0].max := 1.0, [2361].log_data[0].total := 300.0, [2361].log_data[0].time := 300.0, [2361].log_data[0].minminute := 5, [2361].log_data[0].maxminute := 5, [2361].log_data[0].valid := 1, [2361].log_data[1].valid := 1, [2361].log_data[2].valid := 1, [2361].log_data[3].valid := 1, [2361].log_data[4].valid := 1, [2361].log_data[5].valid := 1, [2361].log_data[6].valid := 1, [2361].log_data[7].valid := 1, [2361].log_data[8].valid := 1, [2361].log_data[9].valid := 1, [2361].log_data[10].valid := 1, [2361].log_data[11].valid := 1, [2361].log_data[12].valid := 1, [2361].log_data[13].valid := 1, [2361].log_data[14].valid := 1, [2361].log_data[15].valid := 1, [2361].log_data[16].valid := 1, [2361].log_data[17].valid := 1, [2361].log_data[18].valid := 1, [2361].log_data[19].valid := 1, [2361].time.Year := 2023, [2361].time.Month := 1, [2361].time.Day := 17, [2361].time.Hour := 21, [2361].time.Minute := 9, [2361].time.Second := 59, [2362].log_data[0].min := 1.0, [2362].log_data[0].max := 1.0, [2362].log_data[0].total := 300.0, [2362].log_data[0].time := 300.0, [2362].log_data[0].minminute := 10, [2362].log_data[0].maxminute := 10, [2362].log_data[0].valid := 1, [2362].log_data[1].valid := 1, [2362].log_data[2].valid := 1, [2362].log_data[3].valid := 1, [2362].log_data[4].valid := 1, [2362].log_data[5].valid := 1, [2362].log_data[6].valid := 1, [2362].log_data[7].valid := 1, [2362].log_data[8].valid := 1, [2362].log_data[9].valid := 1, [2362].log_data[10].valid := 1, [2362].log_data[11].valid := 1, [2362].log_data[12].valid := 1, [2362].log_data[13].valid := 1, [2362].log_data[14].valid := 1, [2362].log_data[15].valid := 1, [2362].log_data[16].valid := 1, [2362].log_data[17].valid := 1, [2362].log_data[18].valid := 1, [2362].log_data[19].valid := 1, [2362].time.Year := 2023, [2362].time.Month := 1,
        [2362].time.Day := 17, [2362].time.Hour := 21, [2362].time.Minute := 14, [2362].time.Second := 59, [2363].log_data[0].min := 1.0, [2363].log_data[0].max := 1.0, [2363].log_data[0].total := 300.0, [2363].log_data[0].time := 300.0, [2363].log_data[0].minminute := 15, [2363].log_data[0].maxminute := 15, [2363].log_data[0].valid := 1, [2363].log_data[1].valid := 1, [2363].log_data[2].valid := 1, [2363].log_data[3].valid := 1, [2363].log_data[4].valid := 1, [2363].log_data[5].valid := 1, [2363].log_data[6].valid := 1, [2363].log_data[7].valid := 1, [2363].log_data[8].valid := 1, [2363].log_data[9].valid := 1, [2363].log_data[10].valid := 1, [2363].log_data[11].valid := 1, [2363].log_data[12].valid := 1, [2363].log_data[13].valid := 1, [2363].log_data[14].valid := 1, [2363].log_data[15].valid := 1, [2363].log_data[16].valid := 1, [2363].log_data[17].valid := 1, [2363].log_data[18].valid := 1, [2363].log_data[19].valid := 1, [2363].time.Year := 2023, [2363].time.Month := 1, [2363].time.Day := 17, [2363].time.Hour := 21, [2363].time.Minute := 19, [2363].time.Second := 59, [2364].log_data[0].min := 1.0, [2364].log_data[0].max := 1.0, [2364].log_data[0].total := 300.0, [2364].log_data[0].time := 300.0, [2364].log_data[0].minminute := 20, [2364].log_data[0].maxminute := 20, [2364].log_data[0].valid := 1, [2364].log_data[1].valid := 1, [2364].log_data[2].valid := 1, [2364].log_data[3].valid := 1, [2364].log_data[4].valid := 1, [2364].log_data[5].valid := 1, [2364].log_data[6].valid := 1, [2364].log_data[7].valid := 1, [2364].log_data[8].valid := 1, [2364].log_data[9].valid := 1, [2364].log_data[10].valid := 1, [2364].log_data[11].valid := 1, [2364].log_data[12].valid := 1, [2364].log_data[13].valid := 1, [2364].log_data[14].valid := 1, [2364].log_data[15].valid := 1, [2364].log_data[16].valid := 1, [2364].log_data[17].valid := 1,
        [2364].log_data[18].valid := 1, [2364].log_data[19].valid := 1, [2364].time.Year := 2023, [2364].time.Month := 1, [2364].time.Day := 17, [2364].time.Hour := 21, [2364].time.Minute := 24, [2364].time.Second := 59, [2365].log_data[0].min := 1.0, [2365].log_data[0].max := 1.0, [2365].log_data[0].total := 300.0, [2365].log_data[0].time := 300.0, [2365].log_data[0].minminute := 25, [2365].log_data[0].maxminute := 25, [2365].log_data[0].valid := 1, [2365].log_data[1].valid := 1, [2365].log_data[2].valid := 1, [2365].log_data[3].valid := 1, [2365].log_data[4].valid := 1, [2365].log_data[5].valid := 1, [2365].log_data[6].valid := 1, [2365].log_data[7].valid := 1, [2365].log_data[8].valid := 1, [2365].log_data[9].valid := 1, [2365].log_data[10].valid := 1, [2365].log_data[11].valid := 1, [2365].log_data[12].valid := 1, [2365].log_data[13].valid := 1, [2365].log_data[14].valid := 1, [2365].log_data[15].valid := 1, [2365].log_data[16].valid := 1, [2365].log_data[17].valid := 1, [2365].log_data[18].valid := 1, [2365].log_data[19].valid := 1, [2365].time.Year := 2023, [2365].time.Month := 1, [2365].time.Day := 17, [2365].time.Hour := 21, [2365].time.Minute := 29, [2365].time.Second := 59, [2366].log_data[0].min := 1.0, [2366].log_data[0].max := 1.0, [2366].log_data[0].total := 300.0, [2366].log_data[0].time := 300.0, [2366].log_data[0].minminute := 30, [2366].log_data[0].maxminute := 30, [2366].log_data[0].valid := 1, [2366].log_data[1].valid := 1, [2366].log_data[2].valid := 1, [2366].log_data[3].valid := 1, [2366].log_data[4].valid := 1, [2366].log_data[5].valid := 1, [2366].log_data[6].valid := 1, [2366].log_data[7].valid := 1, [2366].log_data[8].valid := 1, [2366].log_data[9].valid := 1, [2366].log_data[10].valid := 1, [2366].log_data[11].valid := 1, [2366].log_data[12].valid := 1, [2366].log_data[13].valid := 1,
        [2366].log_data[14].valid := 1, [2366].log_data[15].valid := 1, [2366].log_data[16].valid := 1, [2366].log_data[17].valid := 1, [2366].log_data[18].valid := 1, [2366].log_data[19].valid := 1, [2366].time.Year := 2023, [2366].time.Month := 1, [2366].time.Day := 17, [2366].time.Hour := 21, [2366].time.Minute := 34, [2366].time.Second := 59, [2367].log_data[0].min := 1.0, [2367].log_data[0].max := 1.0, [2367].log_data[0].total := 300.0, [2367].log_data[0].time := 300.0, [2367].log_data[0].minminute := 35, [2367].log_data[0].maxminute := 35, [2367].log_data[0].valid := 1, [2367].log_data[1].valid := 1, [2367].log_data[2].valid := 1, [2367].log_data[3].valid := 1, [2367].log_data[4].valid := 1, [2367].log_data[5].valid := 1, [2367].log_data[6].valid := 1, [2367].log_data[7].valid := 1, [2367].log_data[8].valid := 1, [2367].log_data[9].valid := 1, [2367].log_data[10].valid := 1, [2367].log_data[11].valid := 1, [2367].log_data[12].valid := 1, [2367].log_data[13].valid := 1, [2367].log_data[14].valid := 1, [2367].log_data[15].valid := 1, [2367].log_data[16].valid := 1, [2367].log_data[17].valid := 1, [2367].log_data[18].valid := 1, [2367].log_data[19].valid := 1, [2367].time.Year := 2023, [2367].time.Month := 1, [2367].time.Day := 17, [2367].time.Hour := 21, [2367].time.Minute := 39, [2367].time.Second := 59, [2368].log_data[0].min := 1.0, [2368].log_data[0].max := 1.0, [2368].log_data[0].total := 300.0, [2368].log_data[0].time := 300.0, [2368].log_data[0].minminute := 40, [2368].log_data[0].maxminute := 40, [2368].log_data[0].valid := 1, [2368].log_data[1].valid := 1, [2368].log_data[2].valid := 1, [2368].log_data[3].valid := 1, [2368].log_data[4].valid := 1, [2368].log_data[5].valid := 1, [2368].log_data[6].valid := 1, [2368].log_data[7].valid := 1, [2368].log_data[8].valid := 1, [2368].log_data[9].valid := 1,
        [2368].log_data[10].valid := 1, [2368].log_data[11].valid := 1, [2368].log_data[12].valid := 1, [2368].log_data[13].valid := 1, [2368].log_data[14].valid := 1, [2368].log_data[15].valid := 1, [2368].log_data[16].valid := 1, [2368].log_data[17].valid := 1, [2368].log_data[18].valid := 1, [2368].log_data[19].valid := 1, [2368].time.Year := 2023, [2368].time.Month := 1, [2368].time.Day := 17, [2368].time.Hour := 21, [2368].time.Minute := 44, [2368].time.Second := 59, [2369].log_data[0].min := 1.0, [2369].log_data[0].max := 1.0, [2369].log_data[0].total := 300.0, [2369].log_data[0].time := 300.0, [2369].log_data[0].minminute := 45, [2369].log_data[0].maxminute := 45, [2369].log_data[0].valid := 1, [2369].log_data[1].valid := 1, [2369].log_data[2].valid := 1, [2369].log_data[3].valid := 1, [2369].log_data[4].valid := 1, [2369].log_data[5].valid := 1, [2369].log_data[6].valid := 1, [2369].log_data[7].valid := 1, [2369].log_data[8].valid := 1, [2369].log_data[9].valid := 1, [2369].log_data[10].valid := 1, [2369].log_data[11].valid := 1, [2369].log_data[12].valid := 1, [2369].log_data[13].valid := 1, [2369].log_data[14].valid := 1, [2369].log_data[15].valid := 1, [2369].log_data[16].valid := 1, [2369].log_data[17].valid := 1, [2369].log_data[18].valid := 1, [2369].log_data[19].valid := 1, [2369].time.Year := 2023, [2369].time.Month := 1, [2369].time.Day := 17, [2369].time.Hour := 21, [2369].time.Minute := 49, [2369].time.Second := 59, [2370].log_data[0].min := 1.0, [2370].log_data[0].max := 1.0, [2370].log_data[0].total := 300.0, [2370].log_data[0].time := 300.0, [2370].log_data[0].minminute := 50, [2370].log_data[0].maxminute := 50, [2370].log_data[0].valid := 1, [2370].log_data[1].valid := 1, [2370].log_data[2].valid := 1, [2370].log_data[3].valid := 1, [2370].log_data[4].valid := 1, [2370].log_data[5].valid := 1,
        [2370].log_data[6].valid := 1, [2370].log_data[7].valid := 1, [2370].log_data[8].valid := 1, [2370].log_data[9].valid := 1, [2370].log_data[10].valid := 1, [2370].log_data[11].valid := 1, [2370].log_data[12].valid := 1, [2370].log_data[13].valid := 1, [2370].log_data[14].valid := 1, [2370].log_data[15].valid := 1, [2370].log_data[16].valid := 1, [2370].log_data[17].valid := 1, [2370].log_data[18].valid := 1, [2370].log_data[19].valid := 1, [2370].time.Year := 2023, [2370].time.Month := 1, [2370].time.Day := 17, [2370].time.Hour := 21, [2370].time.Minute := 54, [2370].time.Second := 59, [2371].log_data[0].min := 1.0, [2371].log_data[0].max := 1.0, [2371].log_data[0].total := 300.0, [2371].log_data[0].time := 300.0, [2371].log_data[0].minminute := 55, [2371].log_data[0].maxminute := 55, [2371].log_data[0].valid := 1, [2371].log_data[1].valid := 1, [2371].log_data[2].valid := 1, [2371].log_data[3].valid := 1, [2371].log_data[4].valid := 1, [2371].log_data[5].valid := 1, [2371].log_data[6].valid := 1, [2371].log_data[7].valid := 1, [2371].log_data[8].valid := 1, [2371].log_data[9].valid := 1, [2371].log_data[10].valid := 1, [2371].log_data[11].valid := 1, [2371].log_data[12].valid := 1, [2371].log_data[13].valid := 1, [2371].log_data[14].valid := 1, [2371].log_data[15].valid := 1, [2371].log_data[16].valid := 1, [2371].log_data[17].valid := 1, [2371].log_data[18].valid := 1, [2371].log_data[19].valid := 1, [2371].time.Year := 2023, [2371].time.Month := 1, [2371].time.Day := 17, [2371].time.Hour := 21, [2371].time.Minute := 59, [2371].time.Second := 59, [2372].log_data[0].min := 1.0, [2372].log_data[0].max := 1.0, [2372].log_data[0].total := 300.0, [2372].log_data[0].time := 300.0, [2372].log_data[0].valid := 1, [2372].log_data[1].valid := 1, [2372].log_data[2].valid := 1, [2372].log_data[3].valid := 1,
        [2372].log_data[4].valid := 1, [2372].log_data[5].valid := 1, [2372].log_data[6].valid := 1, [2372].log_data[7].valid := 1, [2372].log_data[8].valid := 1, [2372].log_data[9].valid := 1, [2372].log_data[10].valid := 1, [2372].log_data[11].valid := 1, [2372].log_data[12].valid := 1, [2372].log_data[13].valid := 1, [2372].log_data[14].valid := 1, [2372].log_data[15].valid := 1, [2372].log_data[16].valid := 1, [2372].log_data[17].valid := 1, [2372].log_data[18].valid := 1, [2372].log_data[19].valid := 1, [2372].time.Year := 2023, [2372].time.Month := 1, [2372].time.Day := 17, [2372].time.Hour := 22, [2372].time.Minute := 4, [2372].time.Second := 59, [2373].log_data[0].min := 1.0, [2373].log_data[0].max := 1.0, [2373].log_data[0].total := 300.0, [2373].log_data[0].time := 300.0, [2373].log_data[0].minminute := 5, [2373].log_data[0].maxminute := 5, [2373].log_data[0].valid := 1, [2373].log_data[1].valid := 1, [2373].log_data[2].valid := 1, [2373].log_data[3].valid := 1, [2373].log_data[4].valid := 1, [2373].log_data[5].valid := 1, [2373].log_data[6].valid := 1, [2373].log_data[7].valid := 1, [2373].log_data[8].valid := 1, [2373].log_data[9].valid := 1, [2373].log_data[10].valid := 1, [2373].log_data[11].valid := 1, [2373].log_data[12].valid := 1, [2373].log_data[13].valid := 1, [2373].log_data[14].valid := 1, [2373].log_data[15].valid := 1, [2373].log_data[16].valid := 1, [2373].log_data[17].valid := 1, [2373].log_data[18].valid := 1, [2373].log_data[19].valid := 1, [2373].time.Year := 2023, [2373].time.Month := 1, [2373].time.Day := 17, [2373].time.Hour := 22, [2373].time.Minute := 9, [2373].time.Second := 59, [2374].log_data[0].min := 1.0, [2374].log_data[0].max := 1.0, [2374].log_data[0].total := 300.0, [2374].log_data[0].time := 300.0, [2374].log_data[0].minminute := 10, [2374].log_data[0].maxminute := 10,
        [2374].log_data[0].valid := 1, [2374].log_data[1].valid := 1, [2374].log_data[2].valid := 1, [2374].log_data[3].valid := 1, [2374].log_data[4].valid := 1, [2374].log_data[5].valid := 1, [2374].log_data[6].valid := 1, [2374].log_data[7].valid := 1, [2374].log_data[8].valid := 1, [2374].log_data[9].valid := 1, [2374].log_data[10].valid := 1, [2374].log_data[11].valid := 1, [2374].log_data[12].valid := 1, [2374].log_data[13].valid := 1, [2374].log_data[14].valid := 1, [2374].log_data[15].valid := 1, [2374].log_data[16].valid := 1, [2374].log_data[17].valid := 1, [2374].log_data[18].valid := 1, [2374].log_data[19].valid := 1, [2374].time.Year := 2023, [2374].time.Month := 1, [2374].time.Day := 17, [2374].time.Hour := 22, [2374].time.Minute := 14, [2374].time.Second := 59, [2375].log_data[0].min := 1.0, [2375].log_data[0].max := 1.0, [2375].log_data[0].total := 300.0, [2375].log_data[0].time := 300.0, [2375].log_data[0].minminute := 15, [2375].log_data[0].maxminute := 15, [2375].log_data[0].valid := 1, [2375].log_data[1].valid := 1, [2375].log_data[2].valid := 1, [2375].log_data[3].valid := 1, [2375].log_data[4].valid := 1, [2375].log_data[5].valid := 1, [2375].log_data[6].valid := 1, [2375].log_data[7].valid := 1, [2375].log_data[8].valid := 1, [2375].log_data[9].valid := 1, [2375].log_data[10].valid := 1, [2375].log_data[11].valid := 1, [2375].log_data[12].valid := 1, [2375].log_data[13].valid := 1, [2375].log_data[14].valid := 1, [2375].log_data[15].valid := 1, [2375].log_data[16].valid := 1, [2375].log_data[17].valid := 1, [2375].log_data[18].valid := 1, [2375].log_data[19].valid := 1, [2375].time.Year := 2023, [2375].time.Month := 1, [2375].time.Day := 17, [2375].time.Hour := 22, [2375].time.Minute := 19, [2375].time.Second := 59, [2376].log_data[0].min := 1.0, [2376].log_data[0].max := 1.0,
        [2376].log_data[0].total := 300.0, [2376].log_data[0].time := 300.0, [2376].log_data[0].minminute := 20, [2376].log_data[0].maxminute := 20, [2376].log_data[0].valid := 1, [2376].log_data[1].valid := 1, [2376].log_data[2].valid := 1, [2376].log_data[3].valid := 1, [2376].log_data[4].valid := 1, [2376].log_data[5].valid := 1, [2376].log_data[6].valid := 1, [2376].log_data[7].valid := 1, [2376].log_data[8].valid := 1, [2376].log_data[9].valid := 1, [2376].log_data[10].valid := 1, [2376].log_data[11].valid := 1, [2376].log_data[12].valid := 1, [2376].log_data[13].valid := 1, [2376].log_data[14].valid := 1, [2376].log_data[15].valid := 1, [2376].log_data[16].valid := 1, [2376].log_data[17].valid := 1, [2376].log_data[18].valid := 1, [2376].log_data[19].valid := 1, [2376].time.Year := 2023, [2376].time.Month := 1, [2376].time.Day := 17, [2376].time.Hour := 22, [2376].time.Minute := 24, [2376].time.Second := 59, [2377].log_data[0].min := 1.0, [2377].log_data[0].max := 1.0, [2377].log_data[0].total := 300.0, [2377].log_data[0].time := 300.0, [2377].log_data[0].minminute := 25, [2377].log_data[0].maxminute := 25, [2377].log_data[0].valid := 1, [2377].log_data[1].valid := 1, [2377].log_data[2].valid := 1, [2377].log_data[3].valid := 1, [2377].log_data[4].valid := 1, [2377].log_data[5].valid := 1, [2377].log_data[6].valid := 1, [2377].log_data[7].valid := 1, [2377].log_data[8].valid := 1, [2377].log_data[9].valid := 1, [2377].log_data[10].valid := 1, [2377].log_data[11].valid := 1, [2377].log_data[12].valid := 1, [2377].log_data[13].valid := 1, [2377].log_data[14].valid := 1, [2377].log_data[15].valid := 1, [2377].log_data[16].valid := 1, [2377].log_data[17].valid := 1, [2377].log_data[18].valid := 1, [2377].log_data[19].valid := 1, [2377].time.Year := 2023, [2377].time.Month := 1, [2377].time.Day := 17, [2377].time.Hour := 22,
        [2377].time.Minute := 29, [2377].time.Second := 59, [2378].log_data[0].min := 1.0, [2378].log_data[0].max := 1.0, [2378].log_data[0].total := 300.0, [2378].log_data[0].time := 300.0, [2378].log_data[0].minminute := 30, [2378].log_data[0].maxminute := 30, [2378].log_data[0].valid := 1, [2378].log_data[1].valid := 1, [2378].log_data[2].valid := 1, [2378].log_data[3].valid := 1, [2378].log_data[4].valid := 1, [2378].log_data[5].valid := 1, [2378].log_data[6].valid := 1, [2378].log_data[7].valid := 1, [2378].log_data[8].valid := 1, [2378].log_data[9].valid := 1, [2378].log_data[10].valid := 1, [2378].log_data[11].valid := 1, [2378].log_data[12].valid := 1, [2378].log_data[13].valid := 1, [2378].log_data[14].valid := 1, [2378].log_data[15].valid := 1, [2378].log_data[16].valid := 1, [2378].log_data[17].valid := 1, [2378].log_data[18].valid := 1, [2378].log_data[19].valid := 1, [2378].time.Year := 2023, [2378].time.Month := 1, [2378].time.Day := 17, [2378].time.Hour := 22, [2378].time.Minute := 34, [2378].time.Second := 59, [2379].log_data[0].min := 1.0, [2379].log_data[0].max := 1.0, [2379].log_data[0].total := 300.0, [2379].log_data[0].time := 300.0, [2379].log_data[0].minminute := 35, [2379].log_data[0].maxminute := 35, [2379].log_data[0].valid := 1, [2379].log_data[1].valid := 1, [2379].log_data[2].valid := 1, [2379].log_data[3].valid := 1, [2379].log_data[4].valid := 1, [2379].log_data[5].valid := 1, [2379].log_data[6].valid := 1, [2379].log_data[7].valid := 1, [2379].log_data[8].valid := 1, [2379].log_data[9].valid := 1, [2379].log_data[10].valid := 1, [2379].log_data[11].valid := 1, [2379].log_data[12].valid := 1, [2379].log_data[13].valid := 1, [2379].log_data[14].valid := 1, [2379].log_data[15].valid := 1, [2379].log_data[16].valid := 1, [2379].log_data[17].valid := 1, [2379].log_data[18].valid := 1, [2379].log_data[19].valid := 1,
        [2379].time.Year := 2023, [2379].time.Month := 1, [2379].time.Day := 17, [2379].time.Hour := 22, [2379].time.Minute := 39, [2379].time.Second := 59, [2380].log_data[0].min := 1.0, [2380].log_data[0].max := 1.0, [2380].log_data[0].total := 300.0, [2380].log_data[0].time := 300.0, [2380].log_data[0].minminute := 40, [2380].log_data[0].maxminute := 40, [2380].log_data[0].valid := 1, [2380].log_data[1].valid := 1, [2380].log_data[2].valid := 1, [2380].log_data[3].valid := 1, [2380].log_data[4].valid := 1, [2380].log_data[5].valid := 1, [2380].log_data[6].valid := 1, [2380].log_data[7].valid := 1, [2380].log_data[8].valid := 1, [2380].log_data[9].valid := 1, [2380].log_data[10].valid := 1, [2380].log_data[11].valid := 1, [2380].log_data[12].valid := 1, [2380].log_data[13].valid := 1, [2380].log_data[14].valid := 1, [2380].log_data[15].valid := 1, [2380].log_data[16].valid := 1, [2380].log_data[17].valid := 1, [2380].log_data[18].valid := 1, [2380].log_data[19].valid := 1, [2380].time.Year := 2023, [2380].time.Month := 1, [2380].time.Day := 17, [2380].time.Hour := 22, [2380].time.Minute := 44, [2380].time.Second := 59, [2381].log_data[0].min := 1.0, [2381].log_data[0].max := 1.0, [2381].log_data[0].total := 300.0, [2381].log_data[0].time := 300.0, [2381].log_data[0].minminute := 45, [2381].log_data[0].maxminute := 45, [2381].log_data[0].valid := 1, [2381].log_data[1].valid := 1, [2381].log_data[2].valid := 1, [2381].log_data[3].valid := 1, [2381].log_data[4].valid := 1, [2381].log_data[5].valid := 1, [2381].log_data[6].valid := 1, [2381].log_data[7].valid := 1, [2381].log_data[8].valid := 1, [2381].log_data[9].valid := 1, [2381].log_data[10].valid := 1, [2381].log_data[11].valid := 1, [2381].log_data[12].valid := 1, [2381].log_data[13].valid := 1, [2381].log_data[14].valid := 1, [2381].log_data[15].valid := 1,
        [2381].log_data[16].valid := 1, [2381].log_data[17].valid := 1, [2381].log_data[18].valid := 1, [2381].log_data[19].valid := 1, [2381].time.Year := 2023, [2381].time.Month := 1, [2381].time.Day := 17, [2381].time.Hour := 22, [2381].time.Minute := 49, [2381].time.Second := 59, [2382].log_data[0].min := 1.0, [2382].log_data[0].max := 1.0, [2382].log_data[0].total := 300.0, [2382].log_data[0].time := 300.0, [2382].log_data[0].minminute := 50, [2382].log_data[0].maxminute := 50, [2382].log_data[0].valid := 1, [2382].log_data[1].valid := 1, [2382].log_data[2].valid := 1, [2382].log_data[3].valid := 1, [2382].log_data[4].valid := 1, [2382].log_data[5].valid := 1, [2382].log_data[6].valid := 1, [2382].log_data[7].valid := 1, [2382].log_data[8].valid := 1, [2382].log_data[9].valid := 1, [2382].log_data[10].valid := 1, [2382].log_data[11].valid := 1, [2382].log_data[12].valid := 1, [2382].log_data[13].valid := 1, [2382].log_data[14].valid := 1, [2382].log_data[15].valid := 1, [2382].log_data[16].valid := 1, [2382].log_data[17].valid := 1, [2382].log_data[18].valid := 1, [2382].log_data[19].valid := 1, [2382].time.Year := 2023, [2382].time.Month := 1, [2382].time.Day := 17, [2382].time.Hour := 22, [2382].time.Minute := 54, [2382].time.Second := 59, [2383].log_data[0].min := 1.0, [2383].log_data[0].max := 1.0, [2383].log_data[0].total := 300.0, [2383].log_data[0].time := 300.0, [2383].log_data[0].minminute := 55, [2383].log_data[0].maxminute := 55, [2383].log_data[0].valid := 1, [2383].log_data[1].valid := 1, [2383].log_data[2].valid := 1, [2383].log_data[3].valid := 1, [2383].log_data[4].valid := 1, [2383].log_data[5].valid := 1, [2383].log_data[6].valid := 1, [2383].log_data[7].valid := 1, [2383].log_data[8].valid := 1, [2383].log_data[9].valid := 1, [2383].log_data[10].valid := 1, [2383].log_data[11].valid := 1,
        [2383].log_data[12].valid := 1, [2383].log_data[13].valid := 1, [2383].log_data[14].valid := 1, [2383].log_data[15].valid := 1, [2383].log_data[16].valid := 1, [2383].log_data[17].valid := 1, [2383].log_data[18].valid := 1, [2383].log_data[19].valid := 1, [2383].time.Year := 2023, [2383].time.Month := 1, [2383].time.Day := 17, [2383].time.Hour := 22, [2383].time.Minute := 59, [2383].time.Second := 59, [2384].log_data[0].min := 1.0, [2384].log_data[0].max := 1.0, [2384].log_data[0].total := 300.0, [2384].log_data[0].time := 300.0, [2384].log_data[0].valid := 1, [2384].log_data[1].valid := 1, [2384].log_data[2].valid := 1, [2384].log_data[3].valid := 1, [2384].log_data[4].valid := 1, [2384].log_data[5].valid := 1, [2384].log_data[6].valid := 1, [2384].log_data[7].valid := 1, [2384].log_data[8].valid := 1, [2384].log_data[9].valid := 1, [2384].log_data[10].valid := 1, [2384].log_data[11].valid := 1, [2384].log_data[12].valid := 1, [2384].log_data[13].valid := 1, [2384].log_data[14].valid := 1, [2384].log_data[15].valid := 1, [2384].log_data[16].valid := 1, [2384].log_data[17].valid := 1, [2384].log_data[18].valid := 1, [2384].log_data[19].valid := 1, [2384].time.Year := 2023, [2384].time.Month := 1, [2384].time.Day := 17, [2384].time.Hour := 23, [2384].time.Minute := 4, [2384].time.Second := 59, [2385].log_data[0].min := 1.0, [2385].log_data[0].max := 1.0, [2385].log_data[0].total := 300.0, [2385].log_data[0].time := 300.0, [2385].log_data[0].minminute := 5, [2385].log_data[0].maxminute := 5, [2385].log_data[0].valid := 1, [2385].log_data[1].valid := 1, [2385].log_data[2].valid := 1, [2385].log_data[3].valid := 1, [2385].log_data[4].valid := 1, [2385].log_data[5].valid := 1, [2385].log_data[6].valid := 1, [2385].log_data[7].valid := 1, [2385].log_data[8].valid := 1, [2385].log_data[9].valid := 1,
        [2385].log_data[10].valid := 1, [2385].log_data[11].valid := 1, [2385].log_data[12].valid := 1, [2385].log_data[13].valid := 1, [2385].log_data[14].valid := 1, [2385].log_data[15].valid := 1, [2385].log_data[16].valid := 1, [2385].log_data[17].valid := 1, [2385].log_data[18].valid := 1, [2385].log_data[19].valid := 1, [2385].time.Year := 2023, [2385].time.Month := 1, [2385].time.Day := 17, [2385].time.Hour := 23, [2385].time.Minute := 9, [2385].time.Second := 59, [2386].log_data[0].min := 1.0, [2386].log_data[0].max := 1.0, [2386].log_data[0].total := 300.0, [2386].log_data[0].time := 300.0, [2386].log_data[0].minminute := 10, [2386].log_data[0].maxminute := 10, [2386].log_data[0].valid := 1, [2386].log_data[1].valid := 1, [2386].log_data[2].valid := 1, [2386].log_data[3].valid := 1, [2386].log_data[4].valid := 1, [2386].log_data[5].valid := 1, [2386].log_data[6].valid := 1, [2386].log_data[7].valid := 1, [2386].log_data[8].valid := 1, [2386].log_data[9].valid := 1, [2386].log_data[10].valid := 1, [2386].log_data[11].valid := 1, [2386].log_data[12].valid := 1, [2386].log_data[13].valid := 1, [2386].log_data[14].valid := 1, [2386].log_data[15].valid := 1, [2386].log_data[16].valid := 1, [2386].log_data[17].valid := 1, [2386].log_data[18].valid := 1, [2386].log_data[19].valid := 1, [2386].time.Year := 2023, [2386].time.Month := 1, [2386].time.Day := 17, [2386].time.Hour := 23, [2386].time.Minute := 14, [2386].time.Second := 59, [2387].log_data[0].min := 1.0, [2387].log_data[0].max := 1.0, [2387].log_data[0].total := 300.0, [2387].log_data[0].time := 300.0, [2387].log_data[0].minminute := 15, [2387].log_data[0].maxminute := 15, [2387].log_data[0].valid := 1, [2387].log_data[1].valid := 1, [2387].log_data[2].valid := 1, [2387].log_data[3].valid := 1, [2387].log_data[4].valid := 1, [2387].log_data[5].valid := 1,
        [2387].log_data[6].valid := 1, [2387].log_data[7].valid := 1, [2387].log_data[8].valid := 1, [2387].log_data[9].valid := 1, [2387].log_data[10].valid := 1, [2387].log_data[11].valid := 1, [2387].log_data[12].valid := 1, [2387].log_data[13].valid := 1, [2387].log_data[14].valid := 1, [2387].log_data[15].valid := 1, [2387].log_data[16].valid := 1, [2387].log_data[17].valid := 1, [2387].log_data[18].valid := 1, [2387].log_data[19].valid := 1, [2387].time.Year := 2023, [2387].time.Month := 1, [2387].time.Day := 17, [2387].time.Hour := 23, [2387].time.Minute := 19, [2387].time.Second := 59, [2388].log_data[0].min := 1.0, [2388].log_data[0].max := 1.0, [2388].log_data[0].total := 300.0, [2388].log_data[0].time := 300.0, [2388].log_data[0].minminute := 20, [2388].log_data[0].maxminute := 20, [2388].log_data[0].valid := 1, [2388].log_data[1].valid := 1, [2388].log_data[2].valid := 1, [2388].log_data[3].valid := 1, [2388].log_data[4].valid := 1, [2388].log_data[5].valid := 1, [2388].log_data[6].valid := 1, [2388].log_data[7].valid := 1, [2388].log_data[8].valid := 1, [2388].log_data[9].valid := 1, [2388].log_data[10].valid := 1, [2388].log_data[11].valid := 1, [2388].log_data[12].valid := 1, [2388].log_data[13].valid := 1, [2388].log_data[14].valid := 1, [2388].log_data[15].valid := 1, [2388].log_data[16].valid := 1, [2388].log_data[17].valid := 1, [2388].log_data[18].valid := 1, [2388].log_data[19].valid := 1, [2388].time.Year := 2023, [2388].time.Month := 1, [2388].time.Day := 17, [2388].time.Hour := 23, [2388].time.Minute := 24, [2388].time.Second := 59, [2389].log_data[0].min := 1.0, [2389].log_data[0].max := 1.0, [2389].log_data[0].total := 300.0, [2389].log_data[0].time := 300.0, [2389].log_data[0].minminute := 25, [2389].log_data[0].maxminute := 25, [2389].log_data[0].valid := 1, [2389].log_data[1].valid := 1,
        [2389].log_data[2].valid := 1, [2389].log_data[3].valid := 1, [2389].log_data[4].valid := 1, [2389].log_data[5].valid := 1, [2389].log_data[6].valid := 1, [2389].log_data[7].valid := 1, [2389].log_data[8].valid := 1, [2389].log_data[9].valid := 1, [2389].log_data[10].valid := 1, [2389].log_data[11].valid := 1, [2389].log_data[12].valid := 1, [2389].log_data[13].valid := 1, [2389].log_data[14].valid := 1, [2389].log_data[15].valid := 1, [2389].log_data[16].valid := 1, [2389].log_data[17].valid := 1, [2389].log_data[18].valid := 1, [2389].log_data[19].valid := 1, [2389].time.Year := 2023, [2389].time.Month := 1, [2389].time.Day := 17, [2389].time.Hour := 23, [2389].time.Minute := 29, [2389].time.Second := 59, [2390].log_data[0].min := 1.0, [2390].log_data[0].max := 1.0, [2390].log_data[0].total := 300.0, [2390].log_data[0].time := 300.0, [2390].log_data[0].minminute := 30, [2390].log_data[0].maxminute := 30, [2390].log_data[0].valid := 1, [2390].log_data[1].valid := 1, [2390].log_data[2].valid := 1, [2390].log_data[3].valid := 1, [2390].log_data[4].valid := 1, [2390].log_data[5].valid := 1, [2390].log_data[6].valid := 1, [2390].log_data[7].valid := 1, [2390].log_data[8].valid := 1, [2390].log_data[9].valid := 1, [2390].log_data[10].valid := 1, [2390].log_data[11].valid := 1, [2390].log_data[12].valid := 1, [2390].log_data[13].valid := 1, [2390].log_data[14].valid := 1, [2390].log_data[15].valid := 1, [2390].log_data[16].valid := 1, [2390].log_data[17].valid := 1, [2390].log_data[18].valid := 1, [2390].log_data[19].valid := 1, [2390].time.Year := 2023, [2390].time.Month := 1, [2390].time.Day := 17, [2390].time.Hour := 23, [2390].time.Minute := 34, [2390].time.Second := 59, [2391].log_data[0].min := 1.0, [2391].log_data[0].max := 1.0, [2391].log_data[0].total := 300.0, [2391].log_data[0].time := 300.0,
        [2391].log_data[0].minminute := 35, [2391].log_data[0].maxminute := 35, [2391].log_data[0].valid := 1, [2391].log_data[1].valid := 1, [2391].log_data[2].valid := 1, [2391].log_data[3].valid := 1, [2391].log_data[4].valid := 1, [2391].log_data[5].valid := 1, [2391].log_data[6].valid := 1, [2391].log_data[7].valid := 1, [2391].log_data[8].valid := 1, [2391].log_data[9].valid := 1, [2391].log_data[10].valid := 1, [2391].log_data[11].valid := 1, [2391].log_data[12].valid := 1, [2391].log_data[13].valid := 1, [2391].log_data[14].valid := 1, [2391].log_data[15].valid := 1, [2391].log_data[16].valid := 1, [2391].log_data[17].valid := 1, [2391].log_data[18].valid := 1, [2391].log_data[19].valid := 1, [2391].time.Year := 2023, [2391].time.Month := 1, [2391].time.Day := 17, [2391].time.Hour := 23, [2391].time.Minute := 39, [2391].time.Second := 59, [2392].log_data[0].min := 1.0, [2392].log_data[0].max := 1.0, [2392].log_data[0].total := 300.0, [2392].log_data[0].time := 300.0, [2392].log_data[0].minminute := 40, [2392].log_data[0].maxminute := 40, [2392].log_data[0].valid := 1, [2392].log_data[1].valid := 1, [2392].log_data[2].valid := 1, [2392].log_data[3].valid := 1, [2392].log_data[4].valid := 1, [2392].log_data[5].valid := 1, [2392].log_data[6].valid := 1, [2392].log_data[7].valid := 1, [2392].log_data[8].valid := 1, [2392].log_data[9].valid := 1, [2392].log_data[10].valid := 1, [2392].log_data[11].valid := 1, [2392].log_data[12].valid := 1, [2392].log_data[13].valid := 1, [2392].log_data[14].valid := 1, [2392].log_data[15].valid := 1, [2392].log_data[16].valid := 1, [2392].log_data[17].valid := 1, [2392].log_data[18].valid := 1, [2392].log_data[19].valid := 1, [2392].time.Year := 2023, [2392].time.Month := 1, [2392].time.Day := 17, [2392].time.Hour := 23, [2392].time.Minute := 44, [2392].time.Second := 59,
        [2393].log_data[0].min := 1.0, [2393].log_data[0].max := 1.0, [2393].log_data[0].total := 300.0, [2393].log_data[0].time := 300.0, [2393].log_data[0].minminute := 45, [2393].log_data[0].maxminute := 45, [2393].log_data[0].valid := 1, [2393].log_data[1].valid := 1, [2393].log_data[2].valid := 1, [2393].log_data[3].valid := 1, [2393].log_data[4].valid := 1, [2393].log_data[5].valid := 1, [2393].log_data[6].valid := 1, [2393].log_data[7].valid := 1, [2393].log_data[8].valid := 1, [2393].log_data[9].valid := 1, [2393].log_data[10].valid := 1, [2393].log_data[11].valid := 1, [2393].log_data[12].valid := 1, [2393].log_data[13].valid := 1, [2393].log_data[14].valid := 1, [2393].log_data[15].valid := 1, [2393].log_data[16].valid := 1, [2393].log_data[17].valid := 1, [2393].log_data[18].valid := 1, [2393].log_data[19].valid := 1, [2393].time.Year := 2023, [2393].time.Month := 1, [2393].time.Day := 17, [2393].time.Hour := 23, [2393].time.Minute := 49, [2393].time.Second := 59, [2394].log_data[0].min := 1.0, [2394].log_data[0].max := 1.0, [2394].log_data[0].total := 300.0, [2394].log_data[0].time := 300.0, [2394].log_data[0].minminute := 50, [2394].log_data[0].maxminute := 50, [2394].log_data[0].valid := 1, [2394].log_data[1].valid := 1, [2394].log_data[2].valid := 1, [2394].log_data[3].valid := 1, [2394].log_data[4].valid := 1, [2394].log_data[5].valid := 1, [2394].log_data[6].valid := 1, [2394].log_data[7].valid := 1, [2394].log_data[8].valid := 1, [2394].log_data[9].valid := 1, [2394].log_data[10].valid := 1, [2394].log_data[11].valid := 1, [2394].log_data[12].valid := 1, [2394].log_data[13].valid := 1, [2394].log_data[14].valid := 1, [2394].log_data[15].valid := 1, [2394].log_data[16].valid := 1, [2394].log_data[17].valid := 1, [2394].log_data[18].valid := 1, [2394].log_data[19].valid := 1, [2394].time.Year := 2023, [2394].time.Month := 1,
        [2394].time.Day := 17, [2394].time.Hour := 23, [2394].time.Minute := 54, [2394].time.Second := 59, [2395].log_data[0].min := 1.0, [2395].log_data[0].max := 1.0, [2395].log_data[0].total := 300.0, [2395].log_data[0].time := 300.0, [2395].log_data[0].minminute := 55, [2395].log_data[0].maxminute := 55, [2395].log_data[0].valid := 1, [2395].log_data[1].valid := 1, [2395].log_data[2].valid := 1, [2395].log_data[3].valid := 1, [2395].log_data[4].valid := 1, [2395].log_data[5].valid := 1, [2395].log_data[6].valid := 1, [2395].log_data[7].valid := 1, [2395].log_data[8].valid := 1, [2395].log_data[9].valid := 1, [2395].log_data[10].valid := 1, [2395].log_data[11].valid := 1, [2395].log_data[12].valid := 1, [2395].log_data[13].valid := 1, [2395].log_data[14].valid := 1, [2395].log_data[15].valid := 1, [2395].log_data[16].valid := 1, [2395].log_data[17].valid := 1, [2395].log_data[18].valid := 1, [2395].log_data[19].valid := 1, [2395].time.Year := 2023, [2395].time.Month := 1, [2395].time.Day := 17, [2395].time.Hour := 23, [2395].time.Minute := 59, [2395].time.Second := 59, [2396].log_data[0].min := 1.0, [2396].log_data[0].max := 1.0, [2396].log_data[0].total := 300.0, [2396].log_data[0].time := 300.0, [2396].log_data[0].valid := 1, [2396].log_data[1].valid := 1, [2396].log_data[2].valid := 1, [2396].log_data[3].valid := 1, [2396].log_data[4].valid := 1, [2396].log_data[5].valid := 1, [2396].log_data[6].valid := 1, [2396].log_data[7].valid := 1, [2396].log_data[8].valid := 1, [2396].log_data[9].valid := 1, [2396].log_data[10].valid := 1, [2396].log_data[11].valid := 1, [2396].log_data[12].valid := 1, [2396].log_data[13].valid := 1, [2396].log_data[14].valid := 1, [2396].log_data[15].valid := 1, [2396].log_data[16].valid := 1, [2396].log_data[17].valid := 1, [2396].log_data[18].valid := 1, [2396].log_data[19].valid := 1,
        [2396].time.Year := 2023, [2396].time.Month := 1, [2396].time.Day := 18, [2396].time.Minute := 4, [2396].time.Second := 59, [2397].log_data[0].min := 1.0, [2397].log_data[0].max := 1.0, [2397].log_data[0].total := 300.0, [2397].log_data[0].time := 300.0, [2397].log_data[0].minminute := 5, [2397].log_data[0].maxminute := 5, [2397].log_data[0].valid := 1, [2397].log_data[1].valid := 1, [2397].log_data[2].valid := 1, [2397].log_data[3].valid := 1, [2397].log_data[4].valid := 1, [2397].log_data[5].valid := 1, [2397].log_data[6].valid := 1, [2397].log_data[7].valid := 1, [2397].log_data[8].valid := 1, [2397].log_data[9].valid := 1, [2397].log_data[10].valid := 1, [2397].log_data[11].valid := 1, [2397].log_data[12].valid := 1, [2397].log_data[13].valid := 1, [2397].log_data[14].valid := 1, [2397].log_data[15].valid := 1, [2397].log_data[16].valid := 1, [2397].log_data[17].valid := 1, [2397].log_data[18].valid := 1, [2397].log_data[19].valid := 1, [2397].time.Year := 2023, [2397].time.Month := 1, [2397].time.Day := 18, [2397].time.Minute := 9, [2397].time.Second := 59, [2398].log_data[0].min := 1.0, [2398].log_data[0].max := 1.0, [2398].log_data[0].total := 300.0, [2398].log_data[0].time := 300.0, [2398].log_data[0].minminute := 10, [2398].log_data[0].maxminute := 10, [2398].log_data[0].valid := 1, [2398].log_data[1].valid := 1, [2398].log_data[2].valid := 1, [2398].log_data[3].valid := 1, [2398].log_data[4].valid := 1, [2398].log_data[5].valid := 1, [2398].log_data[6].valid := 1, [2398].log_data[7].valid := 1, [2398].log_data[8].valid := 1, [2398].log_data[9].valid := 1, [2398].log_data[10].valid := 1, [2398].log_data[11].valid := 1, [2398].log_data[12].valid := 1, [2398].log_data[13].valid := 1, [2398].log_data[14].valid := 1, [2398].log_data[15].valid := 1, [2398].log_data[16].valid := 1, [2398].log_data[17].valid := 1,
        [2398].log_data[18].valid := 1, [2398].log_data[19].valid := 1, [2398].time.Year := 2023, [2398].time.Month := 1, [2398].time.Day := 18, [2398].time.Minute := 14, [2398].time.Second := 59, [2399].log_data[0].min := 1.0, [2399].log_data[0].max := 1.0, [2399].log_data[0].total := 300.0, [2399].log_data[0].time := 300.0, [2399].log_data[0].minminute := 15, [2399].log_data[0].maxminute := 15, [2399].log_data[0].valid := 1, [2399].log_data[1].valid := 1, [2399].log_data[2].valid := 1, [2399].log_data[3].valid := 1, [2399].log_data[4].valid := 1, [2399].log_data[5].valid := 1, [2399].log_data[6].valid := 1, [2399].log_data[7].valid := 1, [2399].log_data[8].valid := 1, [2399].log_data[9].valid := 1, [2399].log_data[10].valid := 1, [2399].log_data[11].valid := 1, [2399].log_data[12].valid := 1, [2399].log_data[13].valid := 1, [2399].log_data[14].valid := 1, [2399].log_data[15].valid := 1, [2399].log_data[16].valid := 1, [2399].log_data[17].valid := 1, [2399].log_data[18].valid := 1, [2399].log_data[19].valid := 1, [2399].time.Year := 2023, [2399].time.Month := 1, [2399].time.Day := 18, [2399].time.Minute := 19, [2399].time.Second := 59);
   report5_row_qty : DINT := 2400;
   report_data : LogRecord[200] := ([0].log_data[0].min := 1.0, [0].log_data[0].max := 1.0, [0].log_data[0].total := 3600.0, [0].log_data[0].time := 3600.0, [0].log_data[0].valid := 1, [0].log_data[1].time := 3600.0, [0].log_data[1].valid := 1, [0].log_data[2].time := 3600.0, [0].log_data[2].valid := 1, [0].log_data[3].time := 3600.0, [0].log_data[3].valid := 1, [0].log_data[4].time := 3600.0, [0].log_data[4].valid := 1, [0].log_data[5].time := 3600.0, [0].log_data[5].valid := 1, [0].log_data[6].time := 3600.0, [0].log_data[6].valid := 1, [0].log_data[7].time := 3600.0, [0].log_data[7].valid := 1, [0].log_data[8].max := 1.0, [0].log_data[8].total := 3380.251, [0].log_data[8].time := 3600.0, [0].log_data[8].minminute := 56, [0].log_data[8].valid := 1, [0].log_data[9].max := 1.0, [0].log_data[9].total := 3380.251, [0].log_data[9].time := 3600.0, [0].log_data[9].minminute := 56, [0].log_data[9].valid := 1, [0].log_data[10].min := 1.0, [0].log_data[10].max := 1.0, [0].log_data[10].total := 3600.0, [0].log_data[10].time := 3600.0, [0].log_data[10].valid := 1, [0].log_data[11].time := 3600.0, [0].log_data[11].valid := 1, [0].log_data[12].min := 1.0, [0].log_data[12].max := 1.0, [0].log_data[12].total := 3600.0, [0].log_data[12].time := 3600.0, [0].log_data[12].valid := 1, [0].log_data[13].min := 1.0, [0].log_data[13].max := 1.0, [0].log_data[13].total := 3600.0, [0].log_data[13].time := 3600.0, [0].log_data[13].valid := 1, [0].log_data[14].time := 3600.0, [0].log_data[14].valid := 1, [0].log_data[15].time := 3600.0, [0].log_data[15].valid := 1, [0].log_data[16].time := 3600.0, [0].log_data[16].valid := 1, [0].log_data[17].min := 1.0, [0].log_data[17].max := 1.0, [0].log_data[17].total := 3600.0, [0].log_data[17].time := 3600.0, [0].log_data[17].valid := 1, [0].log_data[18].time := 3600.0, [0].log_data[18].valid := 1, [0].log_data[19].time := 3600.0,
        [0].log_data[19].valid := 1, [0].log_data[20].time := 3600.0, [0].log_data[20].valid := 1, [0].log_data[21].min := 1.0, [0].log_data[21].max := 1.0, [0].log_data[21].total := 3600.0, [0].log_data[21].time := 3600.0, [0].log_data[21].valid := 1, [0].log_data[22].time := 3600.0, [0].log_data[22].valid := 1, [0].log_data[23].time := 3600.0, [0].log_data[23].valid := 1, [0].log_data[24].time := 3600.0, [0].log_data[24].valid := 1, [0].log_data[25].time := 3600.0, [0].log_data[25].valid := 1, [0].log_data[26].time := 3600.0, [0].log_data[26].valid := 1, [0].log_data[27].time := 3600.0, [0].log_data[27].valid := 1, [0].log_data[28].time := 3600.0, [0].log_data[28].valid := 1, [0].log_data[29].min := 1.0, [0].log_data[29].max := 1.0, [0].log_data[29].total := 3600.0, [0].log_data[29].time := 3600.0, [0].log_data[29].valid := 1, [0].log_data[30].min := 1.0, [0].log_data[30].max := 1.0, [0].log_data[30].total := 3600.0, [0].log_data[30].time := 3600.0, [0].log_data[30].valid := 1, [0].log_data[31].max := 1.0, [0].log_data[31].total := 1350.7471, [0].log_data[31].time := 3600.0, [0].log_data[31].maxminute := 9, [0].log_data[31].valid := 1, [0].log_data[32].max := 1.0, [0].log_data[32].total := 1592.5, [0].log_data[32].time := 3600.0, [0].log_data[32].minminute := 8, [0].log_data[32].valid := 1, [0].log_data[33].time := 3600.0, [0].log_data[33].valid := 1, [0].log_data[34].time := 3600.0, [0].log_data[34].valid := 1, [0].log_data[35].max := 1.0, [0].log_data[35].total := 1629.749, [0].log_data[35].time := 3600.0, [0].log_data[35].maxminute := 2, [0].log_data[35].valid := 1, [0].log_data[36].max := 1.0, [0].log_data[36].total := 1224.998, [0].log_data[36].time := 3600.0, [0].log_data[36].valid := 1, [0].log_data[37].time := 3600.0, [0].log_data[37].valid := 1, [0].log_data[38].time := 3600.0, [0].log_data[38].valid := 1, [0].log_data[39].min := 0.9961195,
        [0].log_data[39].max := 1.0064838, [0].log_data[39].total := 3607.3958, [0].log_data[39].time := 3600.0, [0].log_data[39].minminute := 39, [0].log_data[39].maxminute := 38, [0].log_data[39].valid := 1, [0].log_data[40].min := 7.5588202, [0].log_data[40].max := 7.5835533, [0].log_data[40].total := 27270.684, [0].log_data[40].time := 3600.0, [0].log_data[40].minminute := 14, [0].log_data[40].maxminute := 2, [0].log_data[40].valid := 1, [0].log_data[41].min := 0.0402063, [0].log_data[41].max := 0.0669021, [0].log_data[41].total := 185.39493, [0].log_data[41].time := 3600.0, [0].log_data[41].minminute := 33, [0].log_data[41].maxminute := 36, [0].log_data[41].valid := 1, [0].log_data[42].min := 2.2927027, [0].log_data[42].max := 2.3001225, [0].log_data[42].total := 8264.736, [0].log_data[42].time := 3600.0, [0].log_data[42].minminute := 35, [0].log_data[42].maxminute := 52, [0].log_data[42].valid := 1, [0].log_data[43].min := -0.26000214, [0].log_data[43].max := -0.26000214, [0].log_data[43].total := -935.9732, [0].log_data[43].time := 3600.0, [0].log_data[43].valid := 1, [0].log_data[44].min := -0.30000305, [0].log_data[44].max := -0.27999878, [0].log_data[44].total := -1064.7773, [0].log_data[44].time := 3600.0, [0].log_data[44].valid := 1, [0].log_data[45].time := 3600.0, [0].log_data[45].valid := 1, [0].log_data[46].time := 3600.0, [0].log_data[46].valid := 1, [0].log_data[47].time := 3600.0, [0].log_data[47].valid := 1, [0].log_data[48].min := 6.745114, [0].log_data[48].max := 6.7885337, [0].log_data[48].total := 24326.748, [0].log_data[48].time := 3600.0, [0].log_data[48].minminute := 59, [0].log_data[48].valid := 1, [0].log_data[49].min := 8.742197, [0].log_data[49].max := 9.361496, [0].log_data[49].total := 33220.316, [0].log_data[49].time := 3600.0, [0].log_data[49].maxminute := 51, [0].log_data[49].valid := 1, [0].log_data[50].min := 1.9988544, [0].log_data[50].max := 2.0836523, [0].log_data[50].total := 7352.758, [0].log_data[50].time := 3600.0, [0].log_data[50].minminute := 56,
        [0].log_data[50].maxminute := 59, [0].log_data[50].valid := 1, [0].log_data[51].time := 3600.0, [0].log_data[51].valid := 1, [0].log_data[52].min := -2.9800034, [0].log_data[52].max := 0.11999512, [0].log_data[52].total := -7544.9155, [0].log_data[52].time := 3600.0, [0].log_data[52].minminute := 9, [0].log_data[52].maxminute := 8, [0].log_data[52].valid := 1, [0].log_data[53].min := -2.840004, [0].log_data[53].max := 0.19999695, [0].log_data[53].total := -6902.992, [0].log_data[53].time := 3600.0, [0].log_data[53].minminute := 55, [0].log_data[53].maxminute := 1, [0].log_data[53].valid := 1, [0].log_data[54].max := 0.5345, [0].log_data[54].total := 1168.5892, [0].log_data[54].time := 3600.0, [0].log_data[54].minminute := 8, [0].log_data[54].maxminute := 9, [0].log_data[54].valid := 1, [0].log_data[55].max := 0.542, [0].log_data[55].total := 1131.2971, [0].log_data[55].time := 3600.0, [0].log_data[55].maxminute := 33, [0].log_data[55].valid := 1, [0].log_data[56].min := 0.16032413, [0].log_data[56].max := 0.1607167, [0].log_data[56].total := 577.7366, [0].log_data[56].time := 3600.0, [0].log_data[56].minminute := 1, [0].log_data[56].maxminute := 5, [0].log_data[56].valid := 1, [0].log_data[57].min := 0.3219897, [0].log_data[57].max := 0.32242152, [0].log_data[57].total := 1159.7014, [0].log_data[57].time := 3600.0, [0].log_data[57].minminute := 12, [0].log_data[57].maxminute := 29, [0].log_data[57].valid := 1, [0].log_data[58].time := 3600.0, [0].log_data[58].valid := 1, [0].log_data[59].time := 3600.0, [0].log_data[59].valid := 1, [0].log_data[60].valid := 1, [0].log_data[61].valid := 1, [0].log_data[62].valid := 1, [0].log_data[63].valid := 1, [0].log_data[64].valid := 1, [0].log_data[65].valid := 1, [0].log_data[66].valid := 1, [0].log_data[67].valid := 1, [0].log_data[68].valid := 1, [0].log_data[69].valid := 1, [0].log_data[70].valid := 1, [0].log_data[71].valid := 1, [0].log_data[72].valid := 1,
        [0].log_data[73].valid := 1, [0].log_data[74].valid := 1, [0].log_data[75].valid := 1, [0].log_data[76].valid := 1, [0].log_data[77].valid := 1, [0].log_data[78].valid := 1, [0].log_data[79].valid := 1, [0].log_data[80].valid := 1, [0].log_data[81].valid := 1, [0].log_data[82].valid := 1, [0].log_data[83].valid := 1, [0].log_data[84].valid := 1, [0].log_data[85].valid := 1, [0].log_data[86].valid := 1, [0].log_data[87].valid := 1, [0].log_data[88].valid := 1, [0].log_data[89].valid := 1, [0].log_data[90].valid := 1, [0].log_data[91].valid := 1, [0].log_data[92].valid := 1, [0].log_data[93].valid := 1, [0].log_data[94].valid := 1, [0].log_data[95].valid := 1, [0].log_data[96].valid := 1, [0].log_data[97].valid := 1, [0].log_data[98].valid := 1, [0].log_data[99].valid := 1, [0].log_data[100].valid := 1, [0].log_data[101].valid := 1, [0].log_data[102].valid := 1, [0].log_data[103].valid := 1, [0].log_data[104].valid := 1, [0].log_data[105].valid := 1, [0].log_data[106].valid := 1, [0].log_data[107].valid := 1, [0].log_data[108].valid := 1, [0].log_data[109].valid := 1, [0].log_data[110].valid := 1, [0].log_data[111].valid := 1, [0].log_data[112].valid := 1, [0].log_data[113].valid := 1, [0].log_data[114].valid := 1, [0].log_data[115].valid := 1, [0].log_data[116].valid := 1, [0].log_data[117].valid := 1, [0].log_data[118].valid := 1, [0].log_data[119].valid := 1, [0].log_data[120].valid := 1, [0].log_data[121].valid := 1, [0].log_data[122].valid := 1, [0].log_data[123].valid := 1, [0].log_data[124].valid := 1, [0].time.Year := 2023, [0].time.Month := 1, [0].time.Day := 13, [0].time.Hour := 3, [0].time.Minute := 59, [0].time.Second := 59, [1].log_data[0].min := 1.0, [1].log_data[0].max := 1.0,
        [1].log_data[0].total := 3600.0, [1].log_data[0].time := 3600.0, [1].log_data[0].valid := 1, [1].log_data[1].time := 3600.0, [1].log_data[1].valid := 1, [1].log_data[2].time := 3600.0, [1].log_data[2].valid := 1, [1].log_data[3].time := 3600.0, [1].log_data[3].valid := 1, [1].log_data[4].time := 3600.0, [1].log_data[4].valid := 1, [1].log_data[5].time := 3600.0, [1].log_data[5].valid := 1, [1].log_data[6].time := 3600.0, [1].log_data[6].valid := 1, [1].log_data[7].time := 3600.0, [1].log_data[7].valid := 1, [1].log_data[8].time := 3600.0, [1].log_data[8].valid := 1, [1].log_data[9].time := 3600.0, [1].log_data[9].valid := 1, [1].log_data[10].min := 1.0, [1].log_data[10].max := 1.0, [1].log_data[10].total := 3600.0, [1].log_data[10].time := 3600.0, [1].log_data[10].valid := 1, [1].log_data[11].time := 3600.0, [1].log_data[11].valid := 1, [1].log_data[12].min := 1.0, [1].log_data[12].max := 1.0, [1].log_data[12].total := 3600.0, [1].log_data[12].time := 3600.0, [1].log_data[12].valid := 1, [1].log_data[13].min := 1.0, [1].log_data[13].max := 1.0, [1].log_data[13].total := 3600.0, [1].log_data[13].time := 3600.0, [1].log_data[13].valid := 1, [1].log_data[14].time := 3600.0, [1].log_data[14].valid := 1, [1].log_data[15].time := 3600.0, [1].log_data[15].valid := 1, [1].log_data[16].time := 3600.0, [1].log_data[16].valid := 1, [1].log_data[17].min := 1.0, [1].log_data[17].max := 1.0, [1].log_data[17].total := 3600.0, [1].log_data[17].time := 3600.0, [1].log_data[17].valid := 1, [1].log_data[18].time := 3600.0, [1].log_data[18].valid := 1, [1].log_data[19].time := 3600.0, [1].log_data[19].valid := 1, [1].log_data[20].time := 3600.0, [1].log_data[20].valid := 1, [1].log_data[21].min := 1.0, [1].log_data[21].max := 1.0, [1].log_data[21].total := 3600.0, [1].log_data[21].time := 3600.0, [1].log_data[21].valid := 1,
        [1].log_data[22].time := 3600.0, [1].log_data[22].valid := 1, [1].log_data[23].time := 3600.0, [1].log_data[23].valid := 1, [1].log_data[24].time := 3600.0, [1].log_data[24].valid := 1, [1].log_data[25].time := 3600.0, [1].log_data[25].valid := 1, [1].log_data[26].time := 3600.0, [1].log_data[26].valid := 1, [1].log_data[27].time := 3600.0, [1].log_data[27].valid := 1, [1].log_data[28].time := 3600.0, [1].log_data[28].valid := 1, [1].log_data[29].min := 1.0, [1].log_data[29].max := 1.0, [1].log_data[29].total := 3600.0, [1].log_data[29].time := 3600.0, [1].log_data[29].valid := 1, [1].log_data[30].min := 1.0, [1].log_data[30].max := 1.0, [1].log_data[30].total := 3600.0, [1].log_data[30].time := 3600.0, [1].log_data[30].valid := 1, [1].log_data[31].time := 3600.0, [1].log_data[31].valid := 1, [1].log_data[32].time := 3600.0, [1].log_data[32].valid := 1, [1].log_data[33].time := 3600.0, [1].log_data[33].valid := 1, [1].log_data[34].time := 3600.0, [1].log_data[34].valid := 1, [1].log_data[35].time := 3600.0, [1].log_data[35].valid := 1, [1].log_data[36].time := 3600.0, [1].log_data[36].valid := 1, [1].log_data[37].time := 3600.0, [1].log_data[37].valid := 1, [1].log_data[38].time := 3600.0, [1].log_data[38].valid := 1, [1].log_data[39].min := 0.9957663, [1].log_data[39].max := 1.0067194, [1].log_data[39].total := 3606.1482, [1].log_data[39].time := 3600.0, [1].log_data[39].minminute := 30, [1].log_data[39].maxminute := 55, [1].log_data[39].valid := 1, [1].log_data[40].min := 7.5659657, [1].log_data[40].max := 7.5808053, [1].log_data[40].total := 27271.762, [1].log_data[40].time := 3600.0, [1].log_data[40].minminute := 51, [1].log_data[40].maxminute := 26, [1].log_data[40].valid := 1, [1].log_data[41].min := 0.04432837, [1].log_data[41].max := 0.14797021, [1].log_data[41].total := 200.72943, [1].log_data[41].time := 3600.0, [1].log_data[41].maxminute := 58, [1].log_data[41].valid := 1,
        [1].log_data[42].min := 2.2912893, [1].log_data[42].max := 2.2992978, [1].log_data[42].total := 8264.971, [1].log_data[42].time := 3600.0, [1].log_data[42].minminute := 8, [1].log_data[42].maxminute := 43, [1].log_data[42].valid := 1, [1].log_data[43].min := -0.27999878, [1].log_data[43].max := -0.26000214, [1].log_data[43].total := -935.9782, [1].log_data[43].time := 3600.0, [1].log_data[43].minminute := 17, [1].log_data[43].valid := 1, [1].log_data[44].min := -0.30000305, [1].log_data[44].max := -0.27999878, [1].log_data[44].total := -1041.8187, [1].log_data[44].time := 3600.0, [1].log_data[44].valid := 1, [1].log_data[45].time := 3600.0, [1].log_data[45].valid := 1, [1].log_data[46].time := 3600.0, [1].log_data[46].valid := 1, [1].log_data[47].time := 3600.0, [1].log_data[47].valid := 1, [1].log_data[48].min := 6.7448387, [1].log_data[48].max := 6.759954, [1].log_data[48].total := 24305.084, [1].log_data[48].time := 3600.0, [1].log_data[48].maxminute := 57, [1].log_data[48].valid := 1, [1].log_data[49].min := 9.289064, [1].log_data[49].max := 9.340296, [1].log_data[49].total := 33518.23, [1].log_data[49].time := 3600.0, [1].log_data[49].minminute := 33, [1].log_data[49].maxminute := 59, [1].log_data[49].valid := 1, [1].log_data[50].min := 2.0824747, [1].log_data[50].max := 2.1118004, [1].log_data[50].total := 7576.87, [1].log_data[50].time := 3600.0, [1].log_data[50].maxminute := 47, [1].log_data[50].valid := 1, [1].log_data[51].time := 3600.0, [1].log_data[51].valid := 1, [1].log_data[52].min := -1.5800018, [1].log_data[52].max := -1.1800003, [1].log_data[52].total := -5384.562, [1].log_data[52].time := 3600.0, [1].log_data[52].minminute := 29, [1].log_data[52].valid := 1, [1].log_data[53].min := -1.4400024, [1].log_data[53].max := -1.0999985, [1].log_data[53].total := -4796.1616, [1].log_data[53].time := 3600.0, [1].log_data[53].minminute := 11, [1].log_data[53].valid := 1, [1].log_data[54].time := 3600.0, [1].log_data[54].valid := 1, [1].log_data[55].time := 3600.0,
        [1].log_data[55].valid := 1, [1].log_data[56].min := 0.16032413, [1].log_data[56].max := 0.1607167, [1].log_data[56].total := 577.68896, [1].log_data[56].time := 3600.0, [1].log_data[56].minminute := 7, [1].log_data[56].valid := 1, [1].log_data[57].min := 0.3219897, [1].log_data[57].max := 0.32238227, [1].log_data[57].total := 1159.7108, [1].log_data[57].time := 3600.0, [1].log_data[57].minminute := 18, [1].log_data[57].maxminute := 6, [1].log_data[57].valid := 1, [1].log_data[58].time := 3600.0, [1].log_data[58].valid := 1, [1].log_data[59].time := 3600.0, [1].log_data[59].valid := 1, [1].log_data[60].valid := 1, [1].log_data[61].valid := 1, [1].log_data[62].valid := 1, [1].log_data[63].valid := 1, [1].log_data[64].valid := 1, [1].log_data[65].valid := 1, [1].log_data[66].valid := 1, [1].log_data[67].valid := 1, [1].log_data[68].valid := 1, [1].log_data[69].valid := 1, [1].log_data[70].valid := 1, [1].log_data[71].valid := 1, [1].log_data[72].valid := 1, [1].log_data[73].valid := 1, [1].log_data[74].valid := 1, [1].log_data[75].valid := 1, [1].log_data[76].valid := 1, [1].log_data[77].valid := 1, [1].log_data[78].valid := 1, [1].log_data[79].valid := 1, [1].log_data[80].valid := 1, [1].log_data[81].valid := 1, [1].log_data[82].valid := 1, [1].log_data[83].valid := 1, [1].log_data[84].valid := 1, [1].log_data[85].valid := 1, [1].log_data[86].valid := 1, [1].log_data[87].valid := 1, [1].log_data[88].valid := 1, [1].log_data[89].valid := 1, [1].log_data[90].valid := 1, [1].log_data[91].valid := 1, [1].log_data[92].valid := 1, [1].log_data[93].valid := 1, [1].log_data[94].valid := 1, [1].log_data[95].valid := 1, [1].log_data[96].valid := 1, [1].log_data[97].valid := 1, [1].log_data[98].valid := 1, [1].log_data[99].valid := 1, [1].log_data[100].valid := 1, [1].log_data[101].valid := 1,
        [1].log_data[102].valid := 1, [1].log_data[103].valid := 1, [1].log_data[104].valid := 1, [1].log_data[105].valid := 1, [1].log_data[106].valid := 1, [1].log_data[107].valid := 1, [1].log_data[108].valid := 1, [1].log_data[109].valid := 1, [1].log_data[110].valid := 1, [1].log_data[111].valid := 1, [1].log_data[112].valid := 1, [1].log_data[113].valid := 1, [1].log_data[114].valid := 1, [1].log_data[115].valid := 1, [1].log_data[116].valid := 1, [1].log_data[117].valid := 1, [1].log_data[118].valid := 1, [1].log_data[119].valid := 1, [1].log_data[120].valid := 1, [1].log_data[121].valid := 1, [1].log_data[122].valid := 1, [1].log_data[123].valid := 1, [1].log_data[124].valid := 1, [1].time.Year := 2023, [1].time.Month := 1, [1].time.Day := 13, [1].time.Hour := 4, [1].time.Minute := 59, [1].time.Second := 59, [2].log_data[0].min := 1.0, [2].log_data[0].max := 1.0, [2].log_data[0].total := 3600.0, [2].log_data[0].time := 3600.0, [2].log_data[0].valid := 1, [2].log_data[1].max := 1.0, [2].log_data[1].total := 518.0, [2].log_data[1].time := 3600.0, [2].log_data[1].maxminute := 6, [2].log_data[1].valid := 1, [2].log_data[2].max := 1.0, [2].log_data[2].total := 514.5, [2].log_data[2].time := 3600.0, [2].log_data[2].maxminute := 6, [2].log_data[2].valid := 1, [2].log_data[3].time := 3600.0, [2].log_data[3].valid := 1, [2].log_data[4].time := 3600.0, [2].log_data[4].valid := 1, [2].log_data[5].max := 1.0, [2].log_data[5].total := 232.5, [2].log_data[5].time := 3600.0, [2].log_data[5].maxminute := 8, [2].log_data[5].valid := 1, [2].log_data[6].time := 3600.0, [2].log_data[6].valid := 1, [2].log_data[7].time := 3600.0, [2].log_data[7].valid := 1, [2].log_data[8].max := 1.0, [2].log_data[8].total := 2975.749, [2].log_data[8].time := 3600.0,
        [2].log_data[8].maxminute := 10, [2].log_data[8].valid := 1, [2].log_data[9].max := 1.0, [2].log_data[9].total := 2972.249, [2].log_data[9].time := 3600.0, [2].log_data[9].maxminute := 10, [2].log_data[9].valid := 1, [2].log_data[10].min := 1.0, [2].log_data[10].max := 1.0, [2].log_data[10].total := 3600.0, [2].log_data[10].time := 3600.0, [2].log_data[10].valid := 1, [2].log_data[11].time := 3600.0, [2].log_data[11].valid := 1, [2].log_data[12].min := 1.0, [2].log_data[12].max := 1.0, [2].log_data[12].total := 3600.0, [2].log_data[12].time := 3600.0, [2].log_data[12].valid := 1, [2].log_data[13].min := 1.0, [2].log_data[13].max := 1.0, [2].log_data[13].total := 3600.0, [2].log_data[13].time := 3600.0, [2].log_data[13].valid := 1, [2].log_data[14].time := 3600.0, [2].log_data[14].valid := 1, [2].log_data[15].time := 3600.0, [2].log_data[15].valid := 1, [2].log_data[16].time := 3600.0, [2].log_data[16].valid := 1, [2].log_data[17].min := 1.0, [2].log_data[17].max := 1.0, [2].log_data[17].total := 3600.0, [2].log_data[17].time := 3600.0, [2].log_data[17].valid := 1, [2].log_data[18].time := 3600.0, [2].log_data[18].valid := 1, [2].log_data[19].time := 3600.0, [2].log_data[19].valid := 1, [2].log_data[20].time := 3600.0, [2].log_data[20].valid := 1, [2].log_data[21].min := 1.0, [2].log_data[21].max := 1.0, [2].log_data[21].total := 3600.0, [2].log_data[21].time := 3600.0, [2].log_data[21].valid := 1, [2].log_data[22].time := 3600.0, [2].log_data[22].valid := 1, [2].log_data[23].time := 3600.0, [2].log_data[23].valid := 1, [2].log_data[24].time := 3600.0, [2].log_data[24].valid := 1, [2].log_data[25].time := 3600.0, [2].log_data[25].valid := 1, [2].log_data[26].time := 3600.0, [2].log_data[26].valid := 1, [2].log_data[27].time := 3600.0, [2].log_data[27].valid := 1, [2].log_data[28].time := 3600.0, [2].log_data[28].valid := 1,
